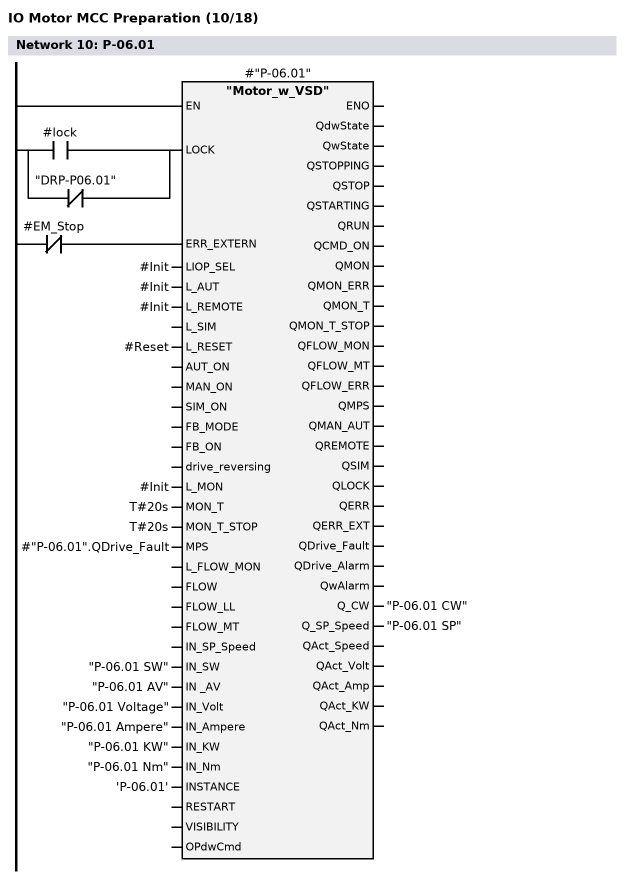
   RUNG wire#powerrail
      #"P-06.01"(LOCK := wire#w1, ERR_EXTERN := wire#w2, LIOP_SEL := #Init, L_AUT := #Init, L_REMOTE := #Init, L_SIM :=, L_RESET := #Reset, AUT_ON :=, MAN_ON :=, SIM_ON :=, FB_MODE :=, FB_ON :=, drive_reversing :=, L_MON := #Init, MON_T := T#20s, MON_T_STOP := T#20s, MPS := #"P-06.01".QDrive_Fault, L_FLOW_MON :=, FLOW :=, FLOW_LL :=, FLOW_MT :=, IN_SP_Speed :=, IN_SW := "P-06.01 SW", "IN _AV" := "P-06.01 AV", IN_Volt := "P-06.01 Voltage", IN_Ampere := "P-06.01 Ampere", IN_KW := "P-06.01 KW", IN_Nm := "P-06.01 Nm", INSTANCE := 'P-06.01', RESTART :=, VISIBILITY :=, OPdwCmd :=, QdwState =>, QwState =>, QSTOPPING =>, QSTOP =>, QSTARTING =>, QRUN =>, QCMD_ON =>, QMON =>, QMON_ERR =>, QMON_T =>, QMON_T_STOP =>, QFLOW_MON =>, QFLOW_MT =>, QFLOW_ERR =>, QMPS =>, QMAN_AUT =>, QREMOTE =>, QSIM =>, QLOCK =>, QERR =>, QERR_EXT =>, QDrive_Fault =>, QDrive_Alarm =>, QwAlarm =>, Q_CW => "P-06.01 CW", Q_SP_Speed => "P-06.01 SP", QAct_Speed =>, QAct_Volt =>, QAct_Amp =>, QAct_KW =>, QAct_Nm =>)
   END_RUNG
   RUNG wire#powerrail
      Contact( #lock )
   END_RUNG wire#w1
   RUNG wire#powerrail
      I_Contact( "DRP-P06.01" )
   END_RUNG wire#w1
   RUNG wire#powerrail
      I_Contact( #EM_Stop )
   END_RUNG wire#w2
   // the same network as SCL:
   #"P-06.01"(LOCK := #lock OR NOT "DRP-P06.01",   // "Motor_w_VSD"
              ERR_EXTERN := NOT #EM_Stop,
              LIOP_SEL := #Init,
              L_AUT := #Init,
              L_REMOTE := #Init,
              L_RESET := #Reset,
              L_MON := #Init,
              MON_T := T#20s,
              MON_T_STOP := T#20s,
              MPS := #"P-06.01".QDrive_Fault,
              IN_SW := "P-06.01 SW",
              "IN _AV" := "P-06.01 AV",
              IN_Volt := "P-06.01 Voltage",
              IN_Ampere := "P-06.01 Ampere",
              IN_KW := "P-06.01 KW",
              IN_Nm := "P-06.01 Nm",
              INSTANCE := 'P-06.01',
              Q_CW => "P-06.01 CW",
              Q_SP_Speed => "P-06.01 SP");
END_REGION

REGION Network 11: P-07.01
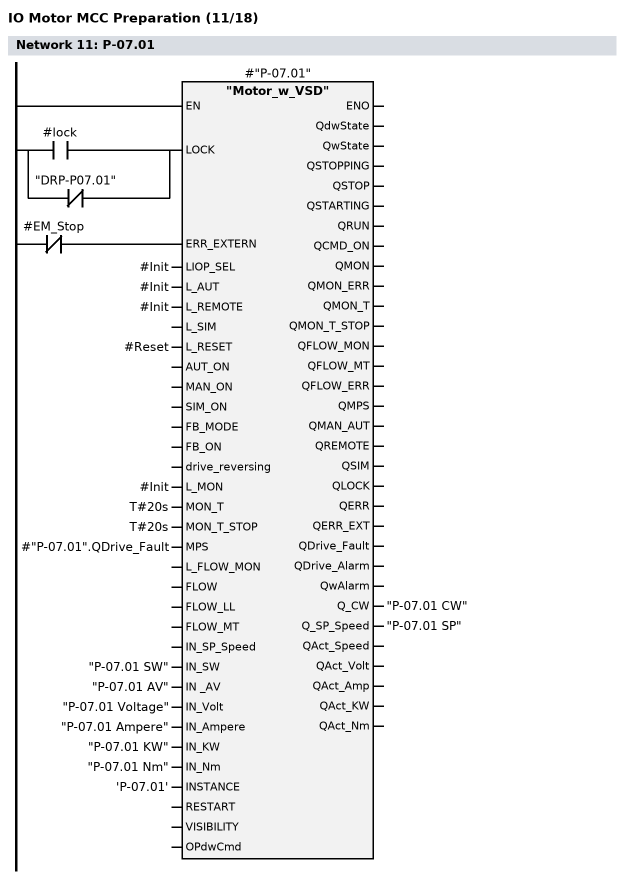
   RUNG wire#powerrail
      #"P-07.01"(LOCK := wire#w1, ERR_EXTERN := wire#w2, LIOP_SEL := #Init, L_AUT := #Init, L_REMOTE := #Init, L_SIM :=, L_RESET := #Reset, AUT_ON :=, MAN_ON :=, SIM_ON :=, FB_MODE :=, FB_ON :=, drive_reversing :=, L_MON := #Init, MON_T := T#20s, MON_T_STOP := T#20s, MPS := #"P-07.01".QDrive_Fault, L_FLOW_MON :=, FLOW :=, FLOW_LL :=, FLOW_MT :=, IN_SP_Speed :=, IN_SW := "P-07.01 SW", "IN _AV" := "P-07.01 AV", IN_Volt := "P-07.01 Voltage", IN_Ampere := "P-07.01 Ampere", IN_KW := "P-07.01 KW", IN_Nm := "P-07.01 Nm", INSTANCE := 'P-07.01', RESTART :=, VISIBILITY :=, OPdwCmd :=, QdwState =>, QwState =>, QSTOPPING =>, QSTOP =>, QSTARTING =>, QRUN =>, QCMD_ON =>, QMON =>, QMON_ERR =>, QMON_T =>, QMON_T_STOP =>, QFLOW_MON =>, QFLOW_MT =>, QFLOW_ERR =>, QMPS =>, QMAN_AUT =>, QREMOTE =>, QSIM =>, QLOCK =>, QERR =>, QERR_EXT =>, QDrive_Fault =>, QDrive_Alarm =>, QwAlarm =>, Q_CW => "P-07.01 CW", Q_SP_Speed => "P-07.01 SP", QAct_Speed =>, QAct_Volt =>, QAct_Amp =>, QAct_KW =>, QAct_Nm =>)
   END_RUNG
   RUNG wire#powerrail
      Contact( #lock )
   END_RUNG wire#w1
   RUNG wire#powerrail
      I_Contact( "DRP-P07.01" )
   END_RUNG wire#w1
   RUNG wire#powerrail
      I_Contact( #EM_Stop )
   END_RUNG wire#w2
   // the same network as SCL:
   #"P-07.01"(LOCK := #lock OR NOT "DRP-P07.01",   // "Motor_w_VSD"
              ERR_EXTERN := NOT #EM_Stop,
              LIOP_SEL := #Init,
              L_AUT := #Init,
              L_REMOTE := #Init,
              L_RESET := #Reset,
              L_MON := #Init,
              MON_T := T#20s,
              MON_T_STOP := T#20s,
              MPS := #"P-07.01".QDrive_Fault,
              IN_SW := "P-07.01 SW",
              "IN _AV" := "P-07.01 AV",
              IN_Volt := "P-07.01 Voltage",
              IN_Ampere := "P-07.01 Ampere",
              IN_KW := "P-07.01 KW",
              IN_Nm := "P-07.01 Nm",
              INSTANCE := 'P-07.01',
              Q_CW => "P-07.01 CW",
              Q_SP_Speed => "P-07.01 SP");
END_REGION

REGION Network 12: P-08.01
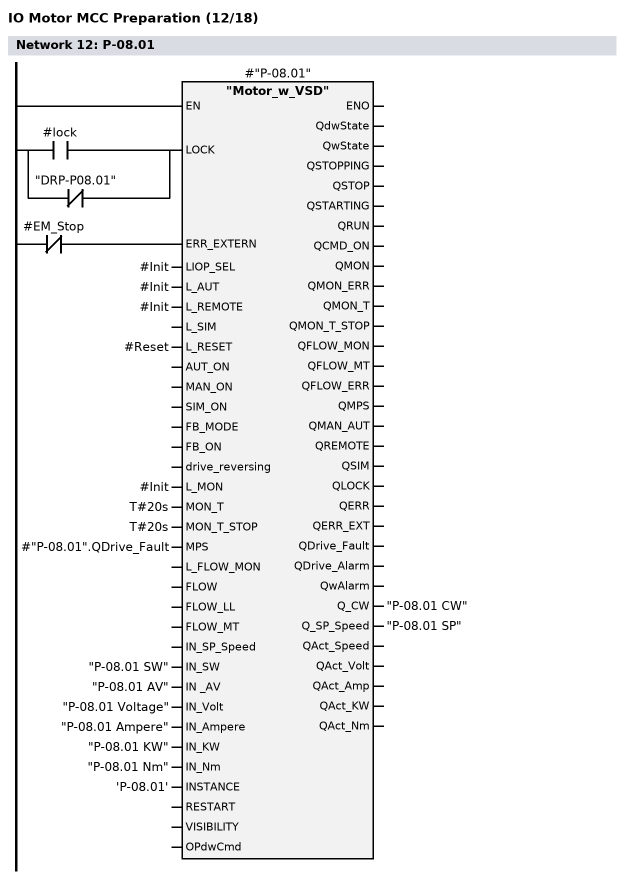
   RUNG wire#powerrail
      #"P-08.01"(LOCK := wire#w1, ERR_EXTERN := wire#w2, LIOP_SEL := #Init, L_AUT := #Init, L_REMOTE := #Init, L_SIM :=, L_RESET := #Reset, AUT_ON :=, MAN_ON :=, SIM_ON :=, FB_MODE :=, FB_ON :=, drive_reversing :=, L_MON := #Init, MON_T := T#20s, MON_T_STOP := T#20s, MPS := #"P-08.01".QDrive_Fault, L_FLOW_MON :=, FLOW :=, FLOW_LL :=, FLOW_MT :=, IN_SP_Speed :=, IN_SW := "P-08.01 SW", "IN _AV" := "P-08.01 AV", IN_Volt := "P-08.01 Voltage", IN_Ampere := "P-08.01 Ampere", IN_KW := "P-08.01 KW", IN_Nm := "P-08.01 Nm", INSTANCE := 'P-08.01', RESTART :=, VISIBILITY :=, OPdwCmd :=, QdwState =>, QwState =>, QSTOPPING =>, QSTOP =>, QSTARTING =>, QRUN =>, QCMD_ON =>, QMON =>, QMON_ERR =>, QMON_T =>, QMON_T_STOP =>, QFLOW_MON =>, QFLOW_MT =>, QFLOW_ERR =>, QMPS =>, QMAN_AUT =>, QREMOTE =>, QSIM =>, QLOCK =>, QERR =>, QERR_EXT =>, QDrive_Fault =>, QDrive_Alarm =>, QwAlarm =>, Q_CW => "P-08.01 CW", Q_SP_Speed => "P-08.01 SP", QAct_Speed =>, QAct_Volt =>, QAct_Amp =>, QAct_KW =>, QAct_Nm =>)
   END_RUNG
   RUNG wire#powerrail
      Contact( #lock )
   END_RUNG wire#w1
   RUNG wire#powerrail
      I_Contact( "DRP-P08.01" )
   END_RUNG wire#w1
   RUNG wire#powerrail
      I_Contact( #EM_Stop )
   END_RUNG wire#w2
   // the same network as SCL:
   #"P-08.01"(LOCK := #lock OR NOT "DRP-P08.01",   // "Motor_w_VSD"
              ERR_EXTERN := NOT #EM_Stop,
              LIOP_SEL := #Init,
              L_AUT := #Init,
              L_REMOTE := #Init,
              L_RESET := #Reset,
              L_MON := #Init,
              MON_T := T#20s,
              MON_T_STOP := T#20s,
              MPS := #"P-08.01".QDrive_Fault,
              IN_SW := "P-08.01 SW",
              "IN _AV" := "P-08.01 AV",
              IN_Volt := "P-08.01 Voltage",
              IN_Ampere := "P-08.01 Ampere",
              IN_KW := "P-08.01 KW",
              IN_Nm := "P-08.01 Nm",
              INSTANCE := 'P-08.01',
              Q_CW => "P-08.01 CW",
              Q_SP_Speed => "P-08.01 SP");
END_REGION

REGION Network 13: P-08.02
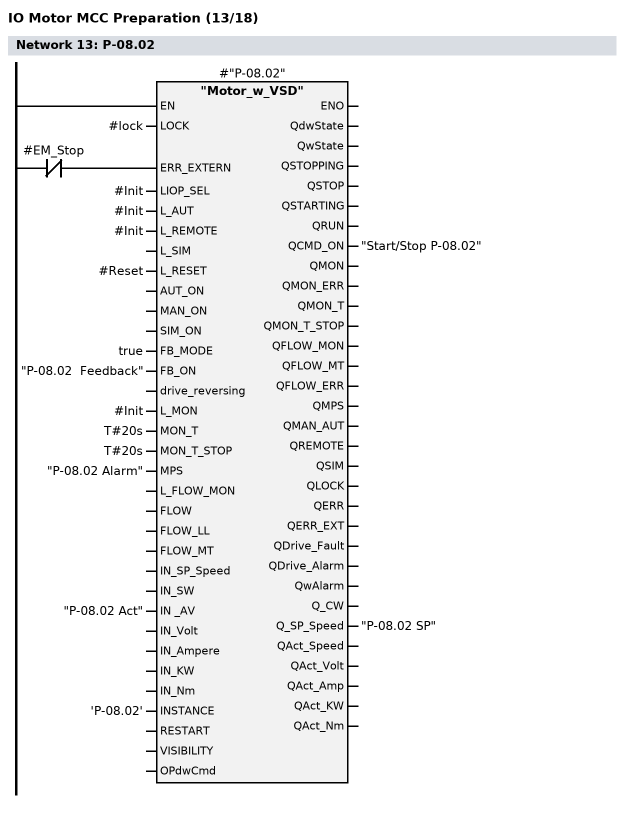
   RUNG wire#powerrail
      #"P-08.02"(ERR_EXTERN := wire#w1, LOCK := #lock, LIOP_SEL := #Init, L_AUT := #Init, L_REMOTE := #Init, L_SIM :=, L_RESET := #Reset, AUT_ON :=, MAN_ON :=, SIM_ON :=, FB_MODE := true, FB_ON := "P-08.02  Feedback", drive_reversing :=, L_MON := #Init, MON_T := T#20s, MON_T_STOP := T#20s, MPS := "P-08.02 Alarm", L_FLOW_MON :=, FLOW :=, FLOW_LL :=, FLOW_MT :=, IN_SP_Speed :=, IN_SW :=, "IN _AV" := "P-08.02 Act", IN_Volt :=, IN_Ampere :=, IN_KW :=, IN_Nm :=, INSTANCE := 'P-08.02', RESTART :=, VISIBILITY :=, OPdwCmd :=, QdwState =>, QwState =>, QSTOPPING =>, QSTOP =>, QSTARTING =>, QRUN =>, QCMD_ON => "Start/Stop P-08.02", QMON =>, QMON_ERR =>, QMON_T =>, QMON_T_STOP =>, QFLOW_MON =>, QFLOW_MT =>, QFLOW_ERR =>, QMPS =>, QMAN_AUT =>, QREMOTE =>, QSIM =>, QLOCK =>, QERR =>, QERR_EXT =>, QDrive_Fault =>, QDrive_Alarm =>, QwAlarm =>, Q_CW =>, Q_SP_Speed => "P-08.02 SP", QAct_Speed =>, QAct_Volt =>, QAct_Amp =>, QAct_KW =>, QAct_Nm =>)
   END_RUNG
   RUNG wire#powerrail
      I_Contact( #EM_Stop )
   END_RUNG wire#w1
   // the same network as SCL:
   #"P-08.02"(LOCK := #lock,   // "Motor_w_VSD"
              ERR_EXTERN := NOT #EM_Stop,
              LIOP_SEL := #Init,
              L_AUT := #Init,
              L_REMOTE := #Init,
              L_RESET := #Reset,
              FB_MODE := true,
              FB_ON := "P-08.02  Feedback",
              L_MON := #Init,
              MON_T := T#20s,
              MON_T_STOP := T#20s,
              MPS := "P-08.02 Alarm",
              "IN _AV" := "P-08.02 Act",
              INSTANCE := 'P-08.02',
              QCMD_ON => "Start/Stop P-08.02",
              Q_SP_Speed => "P-08.02 SP");
END_REGION

REGION Network 14: XA-09.01
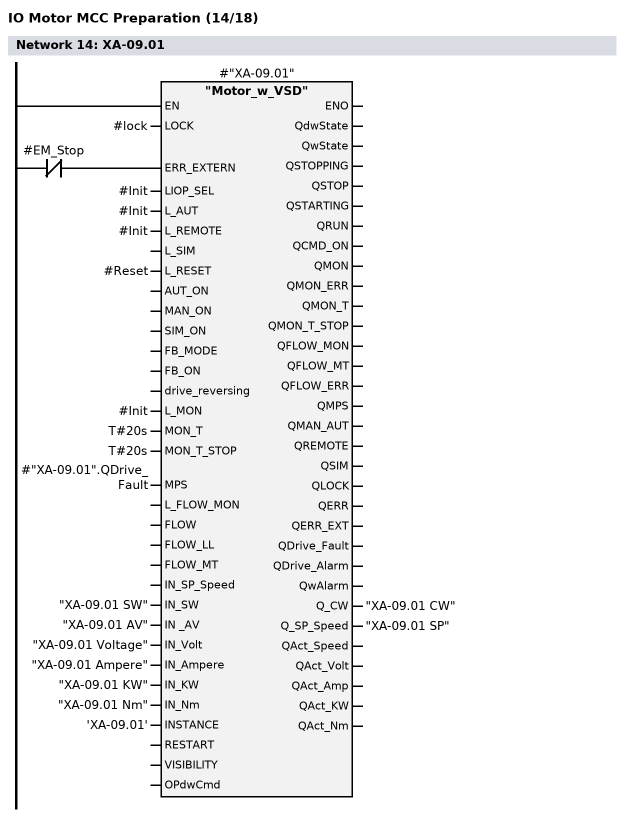
   RUNG wire#powerrail
      #"XA-09.01"(ERR_EXTERN := wire#w1, LOCK := #lock, LIOP_SEL := #Init, L_AUT := #Init, L_REMOTE := #Init, L_SIM :=, L_RESET := #Reset, AUT_ON :=, MAN_ON :=, SIM_ON :=, FB_MODE :=, FB_ON :=, drive_reversing :=, L_MON := #Init, MON_T := T#20s, MON_T_STOP := T#20s, MPS := #"XA-09.01".QDrive_Fault, L_FLOW_MON :=, FLOW :=, FLOW_LL :=, FLOW_MT :=, IN_SP_Speed :=, IN_SW := "XA-09.01 SW", "IN _AV" := "XA-09.01 AV", IN_Volt := "XA-09.01 Voltage", IN_Ampere := "XA-09.01 Ampere", IN_KW := "XA-09.01 KW", IN_Nm := "XA-09.01 Nm", INSTANCE := 'XA-09.01', RESTART :=, VISIBILITY :=, OPdwCmd :=, QdwState =>, QwState =>, QSTOPPING =>, QSTOP =>, QSTARTING =>, QRUN =>, QCMD_ON =>, QMON =>, QMON_ERR =>, QMON_T =>, QMON_T_STOP =>, QFLOW_MON =>, QFLOW_MT =>, QFLOW_ERR =>, QMPS =>, QMAN_AUT =>, QREMOTE =>, QSIM =>, QLOCK =>, QERR =>, QERR_EXT =>, QDrive_Fault =>, QDrive_Alarm =>, QwAlarm =>, Q_CW => "XA-09.01 CW", Q_SP_Speed => "XA-09.01 SP", QAct_Speed =>, QAct_Volt =>, QAct_Amp =>, QAct_KW =>, QAct_Nm =>)
   END_RUNG
   RUNG wire#powerrail
      I_Contact( #EM_Stop )
   END_RUNG wire#w1
   // the same network as SCL:
   #"XA-09.01"(LOCK := #lock,   // "Motor_w_VSD"
               ERR_EXTERN := NOT #EM_Stop,
               LIOP_SEL := #Init,
               L_AUT := #Init,
               L_REMOTE := #Init,
               L_RESET := #Reset,
               L_MON := #Init,
               MON_T := T#20s,
               MON_T_STOP := T#20s,
               MPS := #"XA-09.01".QDrive_Fault,
               IN_SW := "XA-09.01 SW",
               "IN _AV" := "XA-09.01 AV",
               IN_Volt := "XA-09.01 Voltage",
               IN_Ampere := "XA-09.01 Ampere",
               IN_KW := "XA-09.01 KW",
               IN_Nm := "XA-09.01 Nm",
               INSTANCE := 'XA-09.01',
               Q_CW => "XA-09.01 CW",
               Q_SP_Speed => "XA-09.01 SP");
END_REGION

REGION Network 15: P-09.01
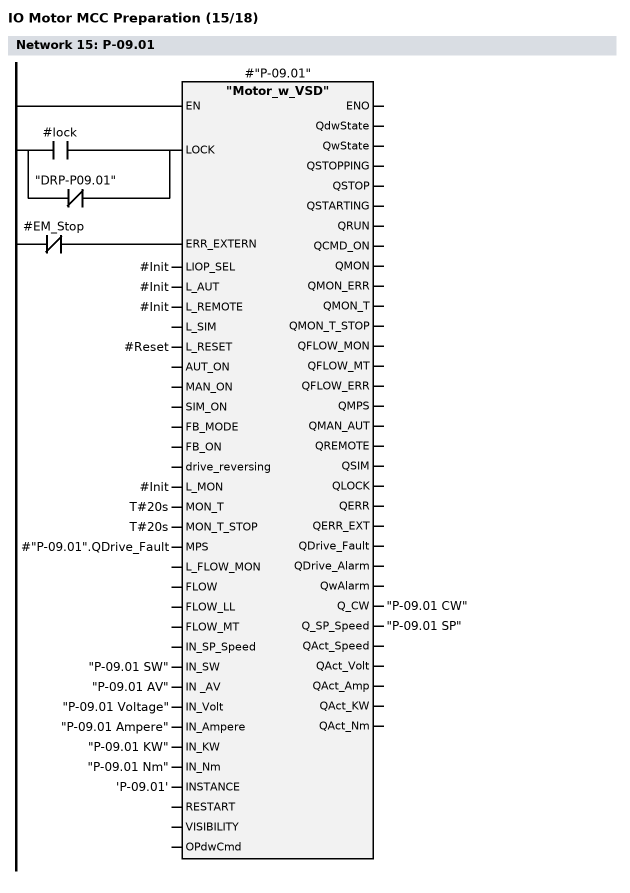
   RUNG wire#powerrail
      #"P-09.01"(LOCK := wire#w1, ERR_EXTERN := wire#w2, LIOP_SEL := #Init, L_AUT := #Init, L_REMOTE := #Init, L_SIM :=, L_RESET := #Reset, AUT_ON :=, MAN_ON :=, SIM_ON :=, FB_MODE :=, FB_ON :=, drive_reversing :=, L_MON := #Init, MON_T := T#20s, MON_T_STOP := T#20s, MPS := #"P-09.01".QDrive_Fault, L_FLOW_MON :=, FLOW :=, FLOW_LL :=, FLOW_MT :=, IN_SP_Speed :=, IN_SW := "P-09.01 SW", "IN _AV" := "P-09.01 AV", IN_Volt := "P-09.01 Voltage", IN_Ampere := "P-09.01 Ampere", IN_KW := "P-09.01 KW", IN_Nm := "P-09.01 Nm", INSTANCE := 'P-09.01', RESTART :=, VISIBILITY :=, OPdwCmd :=, QdwState =>, QwState =>, QSTOPPING =>, QSTOP =>, QSTARTING =>, QRUN =>, QCMD_ON =>, QMON =>, QMON_ERR =>, QMON_T =>, QMON_T_STOP =>, QFLOW_MON =>, QFLOW_MT =>, QFLOW_ERR =>, QMPS =>, QMAN_AUT =>, QREMOTE =>, QSIM =>, QLOCK =>, QERR =>, QERR_EXT =>, QDrive_Fault =>, QDrive_Alarm =>, QwAlarm =>, Q_CW => "P-09.01 CW", Q_SP_Speed => "P-09.01 SP", QAct_Speed =>, QAct_Volt =>, QAct_Amp =>, QAct_KW =>, QAct_Nm =>)
   END_RUNG
   RUNG wire#powerrail
      Contact( #lock )
   END_RUNG wire#w1
   RUNG wire#powerrail
      I_Contact( "DRP-P09.01" )
   END_RUNG wire#w1
   RUNG wire#powerrail
      I_Contact( #EM_Stop )
   END_RUNG wire#w2
   // the same network as SCL:
   #"P-09.01"(LOCK := #lock OR NOT "DRP-P09.01",   // "Motor_w_VSD"
              ERR_EXTERN := NOT #EM_Stop,
              LIOP_SEL := #Init,
              L_AUT := #Init,
              L_REMOTE := #Init,
              L_RESET := #Reset,
              L_MON := #Init,
              MON_T := T#20s,
              MON_T_STOP := T#20s,
              MPS := #"P-09.01".QDrive_Fault,
              IN_SW := "P-09.01 SW",
              "IN _AV" := "P-09.01 AV",
              IN_Volt := "P-09.01 Voltage",
              IN_Ampere := "P-09.01 Ampere",
              IN_KW := "P-09.01 KW",
              IN_Nm := "P-09.01 Nm",
              INSTANCE := 'P-09.01',
              Q_CW => "P-09.01 CW",
              Q_SP_Speed => "P-09.01 SP");
END_REGION

REGION Network 16: P-09.03 DOL
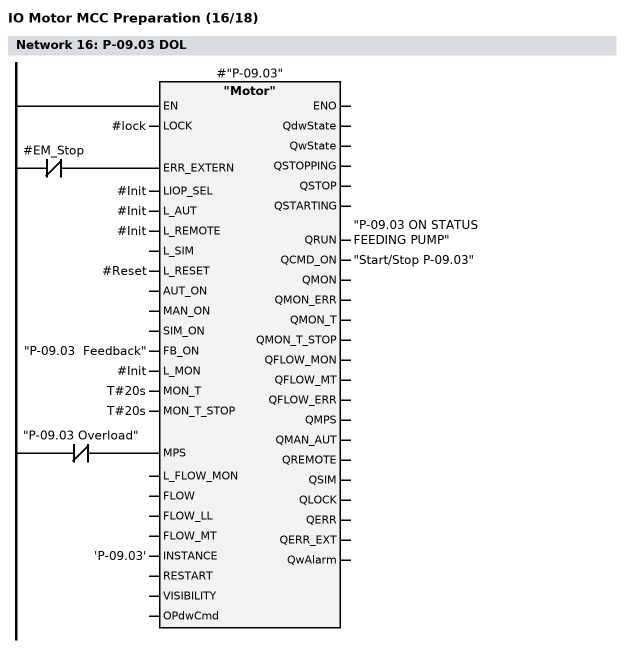
   RUNG wire#powerrail
      #"P-09.03"(ERR_EXTERN := wire#w1, MPS := wire#w2, LOCK := #lock, LIOP_SEL := #Init, L_AUT := #Init, L_REMOTE := #Init, L_SIM :=, L_RESET := #Reset, AUT_ON :=, MAN_ON :=, SIM_ON :=, FB_ON := "P-09.03  Feedback", L_MON := #Init, MON_T := T#20s, MON_T_STOP := T#20s, L_FLOW_MON :=, FLOW :=, FLOW_LL :=, FLOW_MT :=, INSTANCE := 'P-09.03', RESTART :=, VISIBILITY :=, OPdwCmd :=, QdwState =>, QwState =>, QSTOPPING =>, QSTOP =>, QSTARTING =>, QRUN => "P-09.03 ON STATUS FEEDING PUMP", QCMD_ON => "Start/Stop P-09.03", QMON =>, QMON_ERR =>, QMON_T =>, QMON_T_STOP =>, QFLOW_MON =>, QFLOW_MT =>, QFLOW_ERR =>, QMPS =>, QMAN_AUT =>, QREMOTE =>, QSIM =>, QLOCK =>, QERR =>, QERR_EXT =>, QwAlarm =>)
   END_RUNG
   RUNG wire#powerrail
      I_Contact( #EM_Stop )
   END_RUNG wire#w1
   RUNG wire#powerrail
      I_Contact( "P-09.03 Overload" )
   END_RUNG wire#w2
   // the same network as SCL:
   #"P-09.03"(LOCK := #lock,   // "Motor"
              ERR_EXTERN := NOT #EM_Stop,
              LIOP_SEL := #Init,
              L_AUT := #Init,
              L_REMOTE := #Init,
              L_RESET := #Reset,
              FB_ON := "P-09.03  Feedback",
              L_MON := #Init,
              MON_T := T#20s,
              MON_T_STOP := T#20s,
              MPS := NOT "P-09.03 Overload",
              INSTANCE := 'P-09.03',
              QRUN => "P-09.03 ON STATUS FEEDING PUMP",
              QCMD_ON => "Start/Stop P-09.03");
END_REGION

REGION Network 17: P-10.01
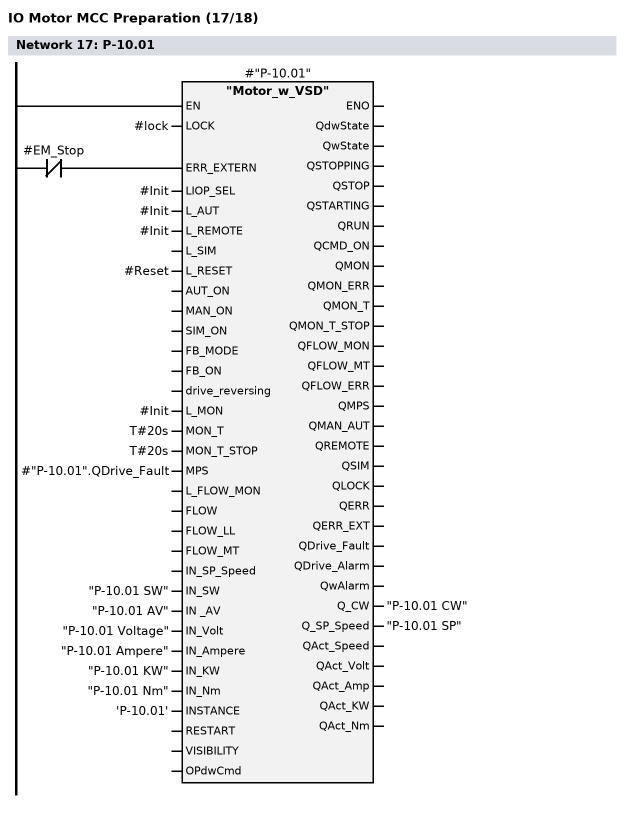
   RUNG wire#powerrail
      #"P-10.01"(ERR_EXTERN := wire#w1, LOCK := #lock, LIOP_SEL := #Init, L_AUT := #Init, L_REMOTE := #Init, L_SIM :=, L_RESET := #Reset, AUT_ON :=, MAN_ON :=, SIM_ON :=, FB_MODE :=, FB_ON :=, drive_reversing :=, L_MON := #Init, MON_T := T#20s, MON_T_STOP := T#20s, MPS := #"P-10.01".QDrive_Fault, L_FLOW_MON :=, FLOW :=, FLOW_LL :=, FLOW_MT :=, IN_SP_Speed :=, IN_SW := "P-10.01 SW", "IN _AV" := "P-10.01 AV", IN_Volt := "P-10.01 Voltage", IN_Ampere := "P-10.01 Ampere", IN_KW := "P-10.01 KW", IN_Nm := "P-10.01 Nm", INSTANCE := 'P-10.01', RESTART :=, VISIBILITY :=, OPdwCmd :=, QdwState =>, QwState =>, QSTOPPING =>, QSTOP =>, QSTARTING =>, QRUN =>, QCMD_ON =>, QMON =>, QMON_ERR =>, QMON_T =>, QMON_T_STOP =>, QFLOW_MON =>, QFLOW_MT =>, QFLOW_ERR =>, QMPS =>, QMAN_AUT =>, QREMOTE =>, QSIM =>, QLOCK =>, QERR =>, QERR_EXT =>, QDrive_Fault =>, QDrive_Alarm =>, QwAlarm =>, Q_CW => "P-10.01 CW", Q_SP_Speed => "P-10.01 SP", QAct_Speed =>, QAct_Volt =>, QAct_Amp =>, QAct_KW =>, QAct_Nm =>)
   END_RUNG
   RUNG wire#powerrail
      I_Contact( #EM_Stop )
   END_RUNG wire#w1
   // the same network as SCL:
   #"P-10.01"(LOCK := #lock,   // "Motor_w_VSD"
              ERR_EXTERN := NOT #EM_Stop,
              LIOP_SEL := #Init,
              L_AUT := #Init,
              L_REMOTE := #Init,
              L_RESET := #Reset,
              L_MON := #Init,
              MON_T := T#20s,
              MON_T_STOP := T#20s,
              MPS := #"P-10.01".QDrive_Fault,
              IN_SW := "P-10.01 SW",
              "IN _AV" := "P-10.01 AV",
              IN_Volt := "P-10.01 Voltage",
              IN_Ampere := "P-10.01 Ampere",
              IN_KW := "P-10.01 KW",
              IN_Nm := "P-10.01 Nm",
              INSTANCE := 'P-10.01',
              Q_CW => "P-10.01 CW",
              Q_SP_Speed => "P-10.01 SP");
END_REGION

REGION Network 18: P-51.01
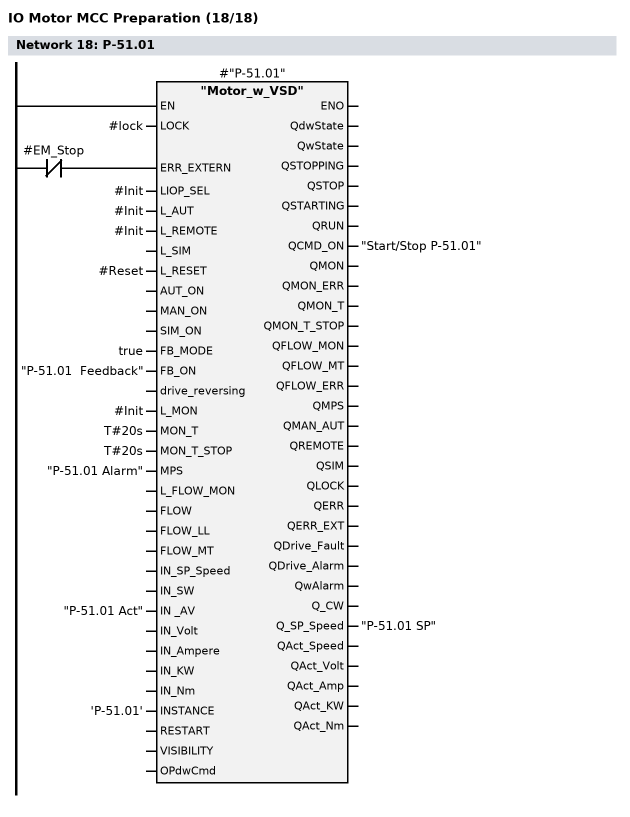
   RUNG wire#powerrail
      #"P-51.01"(ERR_EXTERN := wire#w1, LOCK := #lock, LIOP_SEL := #Init, L_AUT := #Init, L_REMOTE := #Init, L_SIM :=, L_RESET := #Reset, AUT_ON :=, MAN_ON :=, SIM_ON :=, FB_MODE := true, FB_ON := "P-51.01  Feedback", drive_reversing :=, L_MON := #Init, MON_T := T#20s, MON_T_STOP := T#20s, MPS := "P-51.01 Alarm", L_FLOW_MON :=, FLOW :=, FLOW_LL :=, FLOW_MT :=, IN_SP_Speed :=, IN_SW :=, "IN _AV" := "P-51.01 Act", IN_Volt :=, IN_Ampere :=, IN_KW :=, IN_Nm :=, INSTANCE := 'P-51.01', RESTART :=, VISIBILITY :=, OPdwCmd :=, QdwState =>, QwState =>, QSTOPPING =>, QSTOP =>, QSTARTING =>, QRUN =>, QCMD_ON => "Start/Stop P-51.01", QMON =>, QMON_ERR =>, QMON_T =>, QMON_T_STOP =>, QFLOW_MON =>, QFLOW_MT =>, QFLOW_ERR =>, QMPS =>, QMAN_AUT =>, QREMOTE =>, QSIM =>, QLOCK =>, QERR =>, QERR_EXT =>, QDrive_Fault =>, QDrive_Alarm =>, QwAlarm =>, Q_CW =>, Q_SP_Speed => "P-51.01 SP", QAct_Speed =>, QAct_Volt =>, QAct_Amp =>, QAct_KW =>, QAct_Nm =>)
   END_RUNG
   RUNG wire#powerrail
      I_Contact( #EM_Stop )
   END_RUNG wire#w1
   // the same network as SCL:
   #"P-51.01"(LOCK := #lock,   // "Motor_w_VSD"
              ERR_EXTERN := NOT #EM_Stop,
              LIOP_SEL := #Init,
              L_AUT := #Init,
              L_REMOTE := #Init,
              L_RESET := #Reset,
              FB_MODE := true,
              FB_ON := "P-51.01  Feedback",
              L_MON := #Init,
              MON_T := T#20s,
              MON_T_STOP := T#20s,
              MPS := "P-51.01 Alarm",
              "IN _AV" := "P-51.01 Act",
              INSTANCE := 'P-51.01',
              QCMD_ON => "Start/Stop P-51.01",
              Q_SP_Speed => "P-51.01 SP");
END_REGION
END_FUNCTION_BLOCK

FUNCTION_BLOCK "Motor_w_VSD"
TITLE = Motor
{ S7_Optimized_Access := 'FALSE' }
AUTHOR : IW
VERSION : 0.1
//Interface FB for a motor with Danfoss FC Profil
   VAR_INPUT 
      LOCK : Bool;   // 1 = Interlock active
      ERR_EXTERN : Bool;   // 1 = External error arised
      LIOP_SEL : Bool;   // 0 = Operator; 1 = Linking
      L_AUT : Bool;   // 0 = Manual; 1 = Automatic
      L_REMOTE : Bool;   // 0 = Local; 1 = Remote
      L_SIM : Bool;   // 0 = Normal; 1 = Simulation
      L_RESET : Bool;   // 1 = Reset error peripherie
      AUT_ON : Bool;   // 1 = CMD ON Automatic
      MAN_ON : Bool;   // 1 = CMD ON Manual
      SIM_ON : Bool;   // 1 = CMD ON Simulation
      FB_MODE : Bool;   // 0 = FB Run from communication ,1 = FB_ON
      FB_ON : Bool;   // 1 = Feedback Motor ON
      drive_reversing : Bool;
      L_MON : Bool;   // 1 = Monitoring ON
      MON_T : Time := t#5s;   // Monitoring starting time in process mode
      MON_T_STOP : Time := t#5s;   // Monitoring stopping time in process mode
      MPS : Bool;   // 1 = Motor protection switch ON
      L_FLOW_MON : Bool;   // 1 = Monitoring flow
      FLOW : Real;   // Current flow
      FLOW_LL : Real := 5.0;   // Low level flow
      FLOW_MT : Time := t#8s;   // Delay of monitoring lower flow
      IN_SP_Speed : Real;   // Setpoint Speed in Percen
      IN_SW : Word;   // IN Status word from Drive
      "IN _AV" : Int;   // IN Actual Speed from Drive
      IN_Volt : Int;   // IN Actual Voltage
      IN_Ampere : Int;   // IN Actual Ampere
      IN_KW : Int;   // IN Actual KW
      IN_Nm : Int;   // IN Actual Torque
      INSTANCE : String := 'Motor_001';   // Filter attribute for message view, also used for labelling
      RESTART : Bool;   // 1 = Initialize FB at startup (first cycle of PLC)
   END_VAR

   VAR_OUTPUT 
      QdwState : DWord;   // Status HMI
      QwState : Int;   // Motor: 0 = Stop; 1 = Starting; 2 = Run; 3 = Stopping
      QSTOPPING : Bool;   // 1 = Stopping
      QSTOP : Bool;   // 1 = Stop
      QSTARTING : Bool;   // 1 = Starting
      QRUN : Bool;   // 1 = Run
      QCMD_ON : Bool;   // 0 = Stop; 1 = Start (automatic & manual mode)
      QMON : Bool;   // 1 = Monitoring is ON
      QMON_ERR : Bool;   // 1 = Monitoring errror
      QMON_T : Time;   // Expierd starting time in process mode
      QMON_T_STOP : Time;   // Expierd stopping time in process mode
      QFLOW_MON : Bool;   // 1 = Flow monitoring is ON
      QFLOW_MT : Time;   // Expiered delay of monitoring lower flow
      QFLOW_ERR : Bool;   // 1 = Error flow monitoring
      QMPS : Bool;   // 1 = Motor protecting switch
      QMAN_AUT : Bool;   // 0 = Manual; 1 = Automatic
      QREMOTE : Bool;   // 0 = Local; 1 = Remote
      QSIM : Bool;   // 0 = Normal; 1 = Simulation
      QLOCK : Bool;   // 1 = Interlock is active
      QERR : Bool;   // 1 = Common error
      QERR_EXT : Bool;   // 1 = External error
      QDrive_Fault : Bool;
      QDrive_Alarm : Bool;
      QwAlarm : Word;   // Bit alarm procedure
      Q_CW : Word;   // Out Control Word for VSD
      Q_SP_Speed : Word;   // Out SP Speed for VSD
      QAct_Speed : Real;   // Drive Actual Speed
      QAct_Volt : Real;   // Drive Actual Voltage
      QAct_Amp : Real;   // Drive Actual Ampere
      QAct_KW : Real;   // Drive Actual KW
      QAct_Nm : Real;   // Drive Actual Torque
   END_VAR

   VAR_IN_OUT 
      VISIBILITY : Byte;   // Bit 0: Tab1 of window; Bit 1: Tab2 of window; ... ; Bit 7: Minimize
      OPdwCmd : DWord;   // Contorl word HMI
   END_VAR

   VAR 
      FB_SIM : Bool;
      SP_SpeedHz : Real;   // setengah dari 100%
      Drive_Actual_Speed : Real;   // Drive Actual Speed in Percen
      Drive_CW : Word;
      Drive_SW : Word;
      SIM_T : Time;
      QSIM_T : Time;
      SIM_T_STOP : Time;
      QSIM_T_STOP : Time;
      QCMD_SIM : Bool;
      OP_RESET : Bool;   // Reset errors
      QFLOW_MON_ACK : Bool;
      OP_VISIBILITY : Byte;   // Bit 0: Tab1 of window; Bit 1: Tab2 of window; ... ; Bit 7: Minimize
      VISIBILITY_OLD : Byte;   // Save last status of VISIBILITY
      QFB_RUN : Bool;
      Drive_FB_ON : Bool;   // Drive_Running
      Drive_Fault : Bool;   // Drive_Fault Active
      Drive_Alarm : Bool;   // Drive_Alarm Active
      Drive_OK : Bool;
      SE_L_RESET_LINK : Bool;   // Signal edge for the reset input from linking
      SE_L_RESET_LINK_COND : Bool;   // Condition of signal edge
      SE_L_RESET_OP : Bool;   // Signal edge for the reset input from operator
      TSTARTING {InstructionName := 'TON_TIME'; LibVersion := '1.0'} : TON_TIME;
      TSTOPPING {InstructionName := 'TON_TIME'; LibVersion := '1.0'} : TON_TIME;
      TFLOW {InstructionName := 'TON_TIME'; LibVersion := '1.0'} : TON_TIME;
      TSTARTING_SIM {InstructionName := 'TON_TIME'; LibVersion := '1.0'} : TON_TIME;
      TSTOPPING_SIM {InstructionName := 'TON_TIME'; LibVersion := '1.0'} : TON_TIME;
   END_VAR

   VAR_TEMP 
      CON_ERR : Bool;   // Error in motor condition
      MON_ERR_STARTING : Bool;   // Monitoring error for starting motor in process mode
      MON_ERR_STOPPING : Bool;   // Monitoring error for stopping motor in process mode
      MON_SIM_STARTING : Bool;   // Monitoring error for starting motor in simulation mode
      MON_SIM_STOPPING : Bool;   // Monitoring error for stopping motor in simulation mode
      FB_ERR : Bool;   // Feedback error in process mode
      MON_ERR_FLOW2 : Bool;
      START_FLOW_TIME2 : Bool;
      START_FLOW_TIME : Bool;   // Start Signal of delay time for flow
      MON_ERR_FLOW : Bool;   // Monitoring error for flow
   END_VAR


BEGIN
	(********************************
	           Start up
	*********************************)
	IF #RESTART= true THEN
	  // Restart case
	  #QCMD_ON:= false;
	  #QSTOP:=true;
	  #QSTOPPING:=false;
	  #QRUN:=false;
	  #QSTARTING:=false;
	  #VISIBILITY:=0;
	  #OPdwCmd:=0;
	ELSE
	  // Normal case
	  
	  (******************************************
	    Network 1: Operating mode: manual/automatic
	    Vaiable: OPdwCmd  Bit:  16  =  Manual
	    Vaiable: OPdwCmd  Bit:  17  =  Automatic
	  *******************************************)
	  IF (#LIOP_SEL=true AND #L_AUT=true) OR (#OPdwCmd.%X17=true AND #LIOP_SEL=false) THEN
	    #QMAN_AUT:=true;
	    #OPdwCmd.%X16:=false;
	    #OPdwCmd.%X17:=false;
	  ELSIF (#LIOP_SEL=true AND #L_AUT=false) OR (#OPdwCmd.%X16=true AND #LIOP_SEL=false) THEN
	    #QMAN_AUT:= false;
	    #OPdwCmd.%X16:=false;
	    #OPdwCmd.%X17:=false;
	  END_IF;
	  
	  (******************************************
	    Network 2: Control mode: local/remote
	    Vaiable: OPdwCmd  Bit:  18  =  Local
	    Vaiable: OPdwCmd  Bit:  19  =  Remote
	  *******************************************)
	  IF (#LIOP_SEL=true AND #L_REMOTE=true) OR (#OPdwCmd.%X19=true AND #LIOP_SEL=false) THEN
	    #QREMOTE:=true;
	    #OPdwCmd.%X18:=false;
	    #OPdwCmd.%X19:=false;
	  ELSIF (#LIOP_SEL=true AND #L_REMOTE=false) OR (#OPdwCmd.%X18=true AND #LIOP_SEL=false) THEN
	    #QREMOTE:= false;
	    #OPdwCmd.%X18:=false;
	    #OPdwCmd.%X19:=false;
	  END_IF;
	  
	  (******************************************
	    Network 3: Simulation On/Off
	    Vaiable: OPdwCmd  Bit:  20  =  Process
	    Vaiable: OPdwCmd  Bit:  21  =  Simulation
	  *******************************************)
	  IF (#LIOP_SEL=true AND #L_SIM=true) OR (#OPdwCmd.%X21=true AND #LIOP_SEL=false) THEN
	    #QSIM:=true;
	    #OPdwCmd.%X20:=false;
	    #OPdwCmd.%X21:=false;
	  ELSIF (#LIOP_SEL=true AND #L_SIM=false) OR (#OPdwCmd.%X20=true AND #LIOP_SEL=false) THEN
	    #QSIM:= false;
	    #OPdwCmd.%X20:=false;
	    #OPdwCmd.%X21:=false;
	  END_IF;
	  
	  (*************************************
	    Network 4: Reset Operation
	    Vaiable: OPdwCmd  Bit:  24  =  Reset
	  **************************************)
	  // Rising edge by linking
	  IF #L_RESET=true AND #SE_L_RESET_LINK_COND=false THEN
	    #SE_L_RESET_LINK:=true;
	    #SE_L_RESET_LINK_COND:=true;
	  ELSIF #L_RESET=true AND #SE_L_RESET_LINK_COND=true THEN
	    #SE_L_RESET_LINK:=false;
	  ELSE
	    #SE_L_RESET_LINK_COND:=false;
	  END_IF;
	  // Rising edge by operator
	  IF #OPdwCmd.%X24=true THEN
	    #SE_L_RESET_OP:=true;
	    #OPdwCmd.%X24:=false;
	  ELSE
	    #SE_L_RESET_OP:=false;
	  END_IF;
	  // Reset error #OP_RESET:=((#LIOP_SEL AND #SE_L_RESET_LINK) OR (#SE_L_RESET_OP AND NOT #LIOP_SEL)) AND NOT #LOCK;
	  #OP_RESET:=(#L_RESET) OR (#SE_L_RESET_OP AND NOT #LIOP_SEL) AND NOT #LOCK;
	  
	  (**********************************************
	    Network 5: Monitoring feedback ON/OFF
	    Vaiable: OPdwCmd  Bit:  8  =  Monitoring ON
	    Vaiable: OPdwCmd  Bit:  9  =  Monitoring OFF
	  ***********************************************)
	  IF (#LIOP_SEL=true AND #L_MON=false) OR (#OPdwCmd.%X9=true AND #LIOP_SEL=false)THEN
	    #QMON:=false;
	    #OPdwCmd.%X8:=false;
	    #OPdwCmd.%X9:=false;
	  ELSIF (#LIOP_SEL=true AND #L_MON=true) OR (#OPdwCmd.%X8=true AND #LIOP_SEL=false)THEN
	    #QMON:=true;
	    #OPdwCmd.%X8:=false;
	    #OPdwCmd.%X9:=false;
	  END_IF;
	  
	  (***************************************************
	    Network 6: Monitoring flow ON/OFF
	    Vaiable: OPdwCmd  Bit:  10  =  Monitoring flow ON
	    Vaiable: OPdwCmd  Bit:  11  =  Monitoring flow OFF
	  ****************************************************)
	  IF (#LIOP_SEL=true AND #L_FLOW_MON=false) OR (#OPdwCmd.%X11=true AND #LIOP_SEL=false)THEN
	    #QFLOW_MON:=false;
	    #OPdwCmd.%X10:=false;
	    #OPdwCmd.%X11:=false;
	  ELSIF (#LIOP_SEL=true AND #L_FLOW_MON=true) OR (#OPdwCmd.%X10=true AND #LIOP_SEL=false)THEN
	    #QFLOW_MON:=true;
	    #OPdwCmd.%X10:=false;
	    #OPdwCmd.%X11:=false;
	  END_IF;
	  
	   (**********************************************
	    Network 6: START/STOP Motor
	    Vaiable: OPdwCmd  Bit:  0  =  STOP Motor
	    Vaiable: OPdwCmd  Bit:  1  =  START Motor
	  ***********************************************)
	  IF #QERR=false THEN
	    // No errors occurs
	    IF #QSIM=false THEN
	     // Simulation mode is not active
	      // Automatic/Manual mode
	      IF #QMAN_AUT=true THEN
	        // Automatic mode is active
	        // OPEN/CLOSE valve by linking (AUT_ON)
	        #QCMD_ON:=#AUT_ON;
	        #OPdwCmd.%X0:=false;
	        #OPdwCmd.%X1:=false;
	      ELSE
	       // Automatic mode is not active
	        // Local/Remote mode
	        IF #QREMOTE=false THEN
	          // Local mode is active
	          // OPEN/CLOSE valve by linking (MAN_ON)
	          #QCMD_ON:=#MAN_ON AND NOT #QMAN_AUT;
	          #OPdwCmd.%X0:=false;
	          #OPdwCmd.%X1:=false;
	        ELSE
	         // Remote mode is active
	          // Open valve by operator
	          IF #OPdwCmd.%X1=true THEN
	            #QCMD_ON:=true;
	            #OPdwCmd.%X0:=false;
	            #OPdwCmd.%X1:=false;
	          END_IF;
	          // Close valve by operator
	          IF #OPdwCmd.%X0=true THEN
	            #QCMD_ON:=false;
	            #OPdwCmd.%X0:=false;
	            #OPdwCmd.%X1:=false;
	          END_IF;
	        END_IF;
	      END_IF;
	    ELSE
	      // Local/Remote mode
	      IF #QREMOTE=false THEN
	        // Local mode is active
	          // OPEN/CLOSE valve by linking (SIM_ON)
	          #QCMD_SIM:=#SIM_ON;
	          #OPdwCmd.%X0:=false;
	          #OPdwCmd.%X1:=false;
	      ELSE
	        // Remote mode is active
	          // Open valve by operator
	          IF #OPdwCmd.%X1=true THEN
	            #QCMD_SIM:=true;
	            #OPdwCmd.%X0:=false;
	            #OPdwCmd.%X1:=false;
	          END_IF;
	          // Close valve by operator
	          IF #OPdwCmd.%X0=true THEN
	            #QCMD_SIM:=false;
	            #OPdwCmd.%X0:=false;
	            #OPdwCmd.%X1:=false;
	          END_IF;        
	       END_IF;
	    END_IF;  
	  ELSE
	    // Errors occurs
	    #QCMD_ON:=false;
	    #QCMD_SIM:=false;
	    #OPdwCmd.%X0:=false;
	    #OPdwCmd.%X1:=false;
	  END_IF;
	  
	  (****************************************
	    Network 7: Drive FB_Run
	  *****************************************)
	 // #Drive_FB_ON := #IN_SW.%X2 OR ((#IN_SP_Speed < 5.0)AND #QCMD_ON);
	  #Drive_FB_ON := #IN_SW.%X11 OR ((#IN_SP_Speed < 5.0)AND #QCMD_ON);
	  #QFB_RUN := (#FB_MODE = FALSE AND #Drive_FB_ON) OR (#FB_MODE = TRUE AND (#FB_ON OR ((#IN_SP_Speed < 5.0)AND #QCMD_ON)));
	  (****************************************
	    Network 8: Control signal to the Motor (HMI Status)
	  *****************************************)
	  IF #QERR=false THEN
	    // Motor is stopped
	    IF (((#QFB_RUN=false OR #QMON=false) AND #QSIM=false AND #QCMD_ON=false) OR
	      ((#FB_SIM=false OR #QMON=false) AND #QSIM=true AND #QCMD_SIM=false)) AND #QSTOPPING=true THEN
	      #QSTOP:=true;
	      #QSTOPPING:=false;
	      #QRUN:=false;
	      #QSTARTING := false;
	      #QwState:=0;
	    END_IF;
	    // Motor is stopping
	    IF ((#QSIM=false AND #QCMD_ON=false) OR (#QSIM=true AND #QCMD_SIM=false)) AND (#QRUN=true OR #QSTARTING=true) THEN
	      #QSTOP:=false;
	      #QSTOPPING:=true;
	      #QRUN:=false;
	      #QSTARTING:=false;
	      #QwState:=3;
	    END_IF;
	    // Motor is running 
	    IF (((#QFB_RUN=true OR #QMON=false) AND #QSIM=false AND #QCMD_ON=true) OR
	      ((#FB_SIM=true OR #QMON=false) AND #QSIM=true AND #QCMD_SIM=true)) AND #QSTARTING=true THEN    
	    #QSTOP:=false;
	    #QSTOPPING:=false;
	    #QRUN:=true;
	    #QSTARTING:=false;
	    #QwState:=2;
	    END_IF;
	    // Motor is starting 
	    IF ((#QSIM=false AND #QCMD_ON=true) OR (#QSIM=true AND #QCMD_SIM=true)) AND #QSTOP=true THEN
	    #QSTOP:=false;
	    #QSTOPPING:=false;
	    #QRUN:=false;
	    #QSTARTING:=true;
	    #QwState:=1;
	    END_IF;
	  END_IF;
	  (*******************************************************************
	    Network 9: Drive Control Word
	    *******************************************************************)
	  //Drive_OK
	  #Drive_OK := (#IN_SW.%X0 = true AND #IN_SW.%X1 = true) OR
	  (#IN_SW.%X2 = true AND #IN_SW.%X3 = false AND #IN_SW.%X4 = false AND #IN_SW.%X6 = false AND #IN_SW.%X7 = false);
	
	  //Enable PLC Control
	  #Q_CW.%X0 := false;
	  #Q_CW.%X1 := false;
	  #Q_CW.%X2 := true;
	  #Q_CW.%X3 := true;
	  #Q_CW.%X4 := #QCMD_ON = true;   // quick stop
	  #Q_CW.%X5 := true;
	  #Q_CW.%X6 := (#QCMD_ON = true AND #Drive_OK = true);
	  #Q_CW.%X7 := #OP_RESET;
	  #Q_CW.%X8 := false;
	  #Q_CW.%X9 := false;
	  #Q_CW.%X10 := true;
	  #Q_CW.%X11 := false;
	  #Q_CW.%X12 := false;
	  #Q_CW.%X13 := false;
	  #Q_CW.%X14 := false;
	  #Q_CW.%X15 := false;
	  //Drive ON/OFF
	 // IF #QCMD_ON = true THEN
	 //     #Q_CW.%X6 := true;
	 // ELSIF #QCMD_ON = FALSE THEN
	 //     #Q_CW.%X6 := FALSE;
	 // END_IF;
	  //Drive Reversing
	  //IF #drive_reversing = true THEN
	 // #Q_CW.%X11 := true;
	 // ELSIF  #drive_reversing = FALSE THEN
	 //   #Q_CW.%X11 := FALSE;
	 // END_IF;
	//Drive Fault Reset
	 // IF #OP_RESET = true THEN
	 //     #Q_CW.%X7 := true;
	 // ELSIF #OP_RESET = FALSE THEN
	 //     #Q_CW.%X7 := FALSE;
	 // END_IF;
	  (*******************************************************************
	    Network 10: Feedbacks for Running monitoring in process and simulation mode
	  ********************************************************************)
	  IF #QSIM=false AND #QMON=true  THEN
	  // Feedback monitoring in process mode
	    #TSTARTING(IN:=#QSTARTING,
	               PT:=#MON_T,
	               Q=>#MON_ERR_STARTING,
	               ET=>#QMON_T);
	     
	    #TSTOPPING(IN:=#QSTOPPING,
	              PT:=#MON_T_STOP,
	              Q=>#MON_ERR_STOPPING,
	              ET=>#QMON_T_STOP);
	    // Feedback error
	   #FB_ERR := (#QRUN AND NOT #QFB_RUN) OR (#QSTOP AND #QFB_RUN);
	    IF #FB_ERR=true OR #MON_ERR_STARTING=true OR #MON_ERR_STOPPING=true THEN
	      #QMON_ERR:=true;
	    END_IF;
	    
	    
	  ELSIF #QSIM=true AND #QMON=true THEN
	    // Feedback monitoring in simulation mode
	    #TSTARTING_SIM(IN:=#QSTARTING,
	                  PT:=#SIM_T,
	                  Q=>#MON_SIM_STARTING,
	                  ET=>#QSIM_T);
	    
	    #TSTOPPING_SIM(IN:=#QSTOPPING,
	                  PT:=#SIM_T_STOP,
	                  Q=>#MON_SIM_STOPPING,
	                  ET=>#QSIM_T_STOP);
	    
	    // Feedback for start/stop motor in simulation mode
	    IF #MON_SIM_STOPPING=true OR #QERR=true THEN
	      // Feedback for stop
	      #FB_SIM:=false;
	    ELSIF #MON_SIM_STARTING=true THEN
	      // Feedback for start
	      #FB_SIM:=true;
	    END_IF;
	  END_IF;
	
	  (*******************************************************************
	    Network 11: Feedbacks for flow monitoring in process and simulation mode
	  ********************************************************************)
	// Delay time for feedbak flow monitoring
	  #START_FLOW_TIME:=#QFLOW_MON AND (#QSTARTING OR #QRUN) AND NOT #QFLOW_MON_ACK;
	  #TFLOW(IN:=#START_FLOW_TIME,
	         PT:=#FLOW_MT,
	         Q=>#MON_ERR_FLOW,
	         ET=>#QFLOW_MT);
	  
	  //
	  #START_FLOW_TIME2:=false;
	  IF (#FLOW < #FLOW_LL) THEN
	    #START_FLOW_TIME2:=true;
	  END_IF;
	  
	     #TFLOW(IN:=#START_FLOW_TIME2,
	         PT:=#FLOW_MT,
	         Q=>#MON_ERR_FLOW2,
	         ET=>#QFLOW_MT);
	   IF #MON_ERR_FLOW2 THEN
	      #QFLOW_ERR:=true;
	   END_IF;
	  (**********************************************
	    Network 12: Drive Set Speed
	   ***********************************************)
	   //Drive Setpoint Speed in Hz
	   #SP_SpeedHz := #IN_SP_Speed / 2;
	   //Limit Speed 0 to 50 Hz
	   IF #SP_SpeedHz<0.0 THEN
	       GOTO N004;
	   END_IF;
	   IF #SP_SpeedHz > 50.0 THEN
	        GOTO N004;
	    END_IF;
	//OUT = [ ((IN–LO_LIM)/(HI_LIM–LO_LIM)) ∗ (K2–K1) ] + K1
	//UNSCALE Setpoint Speed VSD with hardwire
	//#Q_SP := REAL_TO_INT(((((#IN_SP / 2) - #SP_Lo) / (#SP_Hi - #SP_Lo)) * (#SP_K2 - #SP_K1)) + #SP_K1);
	    IF #FB_MODE = TRUE THEN
	        #Q_SP_Speed := DINT_TO_WORD(ROUND(#SP_SpeedHz * real#100.0) * DINT#27648 / DINT#5000);
	        #Drive_Actual_Speed := (INT_TO_REAL(#"IN _AV") / 27648.0 * 100.0);
	    ELSIF #FB_MODE = FALSE THEN
	        #Q_SP_Speed := DINT_TO_WORD(ROUND(#SP_SpeedHz * real#100.0) * DINT#16384 / DINT#5000);
	        #Drive_Actual_Speed := (INT_TO_REAL(#"IN _AV") / 16354.0 * 100.0);
	    END_IF;
	N004:  ;
	    
	   (**********************************************
	    Network 13: Drive Actual
	  ***********************************************)
	    #QAct_Speed := #Drive_Actual_Speed;
	 //   #QAct_Volt := (INT_TO_REAL(#IN_Volt) / 16354.0 * 1000.0);
	//    #QAct_Amp := (INT_TO_REAL(#IN_Ampere) / 16354.0 * 100.0);
	//    #QAct_KW := (INT_TO_REAL(#IN_KW) / 16354.0 * 100.0);
	//    #QAct_Nm := (INT_TO_REAL(#IN_Nm) / 16354.0 * 100.0);
	
	  (**********************************************
	    Network 14: Check errors
	  ***********************************************)
	   //Drive Fault
	   #QDrive_Fault := #IN_SW.%X3;
	   //Drive Alarm
	   #QDrive_Alarm := #IN_SW.%X7;
	   // External error
	  #QERR_EXT:=#ERR_EXTERN;  
	  // Interlock error
	  IF #LOCK=true AND ( #QSTARTING=true OR #QRUN=true) THEN
	    #QLOCK:=true;
	  END_IF;
	  //
	  IF #MPS=true THEN
	    #QMPS:=true;
	  END_IF;
	  
	  // Error in valve condition
	  #CON_ERR:=NOT((#QSTOP AND NOT #QSTARTING AND NOT #QRUN AND NOT #QSTOPPING) OR
	  (NOT #QSTOP AND #QSTARTING AND NOT #QRUN AND NOT #QSTOPPING) OR
	  (NOT #QSTOP AND NOT #QSTARTING AND #QRUN AND NOT #QSTOPPING) OR
	  (NOT #QSTOP AND NOT #QSTARTING AND NOT #QRUN AND #QSTOPPING));
	
	  (**********************************************
	    Network 15: General error
	  ***********************************************)
	  #QERR:=#QDrive_Fault OR #QDrive_Alarm OR #QERR_EXT OR #QMON_ERR OR #QFLOW_ERR OR #QMPS OR #QLOCK OR #CON_ERR;
	  
	  (**********************************************
	    Network 16: If error then stop
	  ***********************************************)
	  IF #QERR=true THEN
	    #QSTOP:=true;
	    #QSTARTING:=false;
	    #QRUN:=false;
	    #QSTOPPING:=false;
	    #QwState:=0;
	  END_IF;
	  // Reset errors
	  IF #OP_RESET=true THEN
	    #QMON_ERR:=false;
	    #QLOCK:=false;
	    #QFLOW_ERR:=false;
	    #QMPS:=false;
	  END_IF;
	    // End normal case
	END_IF;
	
	(****************************************************
	  Network 13: Influence visibility of faceplate window
	*****************************************************)
	IF #OP_VISIBILITY<>#VISIBILITY_OLD THEN
	  #VISIBILITY_OLD:=#OP_VISIBILITY;
	  #VISIBILITY:=#OP_VISIBILITY;
	ELSIF #VISIBILITY<>#VISIBILITY_OLD THEN
	  #VISIBILITY_OLD:=#VISIBILITY;
	  #OP_VISIBILITY:=#VISIBILITY;
	END_IF;
	(********************************
	  Network 14: Set state for HMI
	*********************************)
	#QdwState.%X0:=#QSTOP AND NOT #QERR;
	#QdwState.%X1:=#QSTARTING;
	#QdwState.%X2:=#QRUN;
	#QdwState.%X3:=#QSTOPPING;
	#QdwState.%X4:=false;
	#QdwState.%X5:=false;
	#QdwState.%X6:=false;
	#QdwState.%X7:=false;
	#QdwState.%X8:=#QMON;
	#QdwState.%X9:=#QMON_ERR;
	#QdwState.%X10:=#QFLOW_MON;
	#QdwState.%X11:=#QFLOW_ERR;
	#QdwState.%X12:=#QMPS;
	#QdwState.%X13:=#QDrive_Fault;
	#QdwState.%X14:=#QDrive_Alarm;
	#QdwState.%X15:=false;
	#QdwState.%X16:=#QMAN_AUT;
	#QdwState.%X17:=#QREMOTE;
	#QdwState.%X18:=#QSIM;
	#QdwState.%X19:=false;
	#QdwState.%X20:=false;
	#QdwState.%X21:=false;
	#QdwState.%X22:=false;
	#QdwState.%X23:=false;
	#QdwState.%X24:=#QERR;
	#QdwState.%X25:=#QERR_EXT;
	#QdwState.%X26:=#QLOCK;
	#QdwState.%X27:=#LOCK;
	#QdwState.%X28:=false;
	#QdwState.%X29:=false;
	#QdwState.%X30:=false;
	#QdwState.%X31:=false;
	
	(********************************
	  Network 15: Bit alarm procedure
	*********************************)
	#QwAlarm.%X0:=#QMON_ERR;
	#QwAlarm.%X1:=#QFLOW_ERR;
	#QwAlarm.%X2:=#MPS;
	#QwAlarm.%X3:=#QDrive_Fault;
	#QwAlarm.%X4:=#QLOCK;
	#QwAlarm.%X5:=#QDrive_Alarm;
	#QwAlarm.%X6:=#QERR_EXT;
	#QwAlarm.%X7:=#QERR;
	#QwAlarm.%X8:=#QSTOP;
	#QwAlarm.%X9:=#QSTARTING;
	#QwAlarm.%X10:=#QRUN;
	#QwAlarm.%X11:=#QSTOPPING;
	#QwAlarm.%X12:=#LOCK;
	#QwAlarm.%X13:=#QREMOTE;
	#QwAlarm.%X14:=#QMAN_AUT;
	#QwAlarm.%X15:=#QSIM;
END_FUNCTION_BLOCK

FUNCTION_BLOCK "Motor"
TITLE = Motor
{ S7_Optimized_Access := 'FALSE' }
AUTHOR : RM
VERSION : 0.1
//Interface FB for a motor
   VAR_INPUT 
      LOCK : Bool;   // 1 = Interlock active
      ERR_EXTERN : Bool;   // 1 = External error arised
      LIOP_SEL : Bool;   // 0 = Operator; 1 = Linking
      L_AUT : Bool;   // 0 = Manual; 1 = Automatic
      L_REMOTE : Bool;   // 0 = Local; 1 = Remote
      L_SIM : Bool;   // 0 = Normal; 1 = Simulation
      L_RESET : Bool;   // 1 = Reset error peripherie
      AUT_ON : Bool;   // 1 = CMD ON Automatic
      MAN_ON : Bool;   // 1 = CMD ON Manual
      SIM_ON : Bool;   // 1 = CMD ON Simulation
      FB_ON : Bool;   // 1 = Feedback Motor ON
      L_MON : Bool;   // 1 = Monitoring ON
      MON_T : Time := t#5s;   // Monitoring starting time in process mode
      MON_T_STOP : Time := t#5s;   // Monitoring stopping time in process mode
      MPS : Bool;   // 1 = Motor protection switch ON
      L_FLOW_MON : Bool;   // 1 = Monitoring flow
      FLOW : Real;   // Current flow
      FLOW_LL : Real := 5.0;   // Low level flow
      FLOW_MT : Time := t#8s;   // Delay of monitoring lower flow
      INSTANCE : String := 'Motor_001';   // Filter attribute for message view, also used for labelling
      RESTART : Bool;   // 1 = Initialize FB at startup (first cycle of PLC)
   END_VAR

   VAR_OUTPUT 
      QdwState : DWord;   // Status HMI
      QwState : Int;   // Motor: 0 = Stop; 1 = Starting; 2 = Run; 3 = Stopping
      QSTOPPING : Bool;   // 1 = Stopping
      QSTOP : Bool;   // 1 = Stop
      QSTARTING : Bool;   // 1 = Starting
      QRUN : Bool;   // 1 = Run
      QCMD_ON : Bool;   // 0 = Stop; 1 = Start (automatic & manual mode)
      QMON : Bool;   // 1 = Monitoring is ON
      QMON_ERR : Bool;   // 1 = Monitoring errror
      QMON_T : Time;   // Expierd starting time in process mode
      QMON_T_STOP : Time;   // Expierd stopping time in process mode
      QFLOW_MON : Bool;   // 1 = Flow monitoring is ON
      QFLOW_MT : Time;   // Expiered delay of monitoring lower flow
      QFLOW_ERR : Bool;   // 1 = Error flow monitoring
      QMPS : Bool;   // 1 = Motor protecting switch
      QMAN_AUT : Bool;   // 0 = Manual; 1 = Automatic
      QREMOTE : Bool;   // 0 = Local; 1 = Remote
      QSIM : Bool;   // 0 = Normal; 1 = Simulation
      QLOCK : Bool;   // 1 = Interlock is active
      QERR : Bool;   // 1 = Common error
      QERR_EXT : Bool;   // 1 = External error
      QwAlarm : Word;   // Bit alarm procedure
   END_VAR

   VAR_IN_OUT 
      VISIBILITY : Byte;   // Bit 0: Tab1 of window; Bit 1: Tab2 of window; ... ; Bit 7: Minimize
      OPdwCmd : DWord;   // Contorl word HMI
   END_VAR

   VAR 
      FB_SIM : Bool;
      SIM_T : Time;
      QSIM_T : Time;
      SIM_T_STOP : Time;
      QSIM_T_STOP : Time;
      QCMD_SIM : Bool;
      OP_RESET : Bool;   // Reset errors
      QFLOW_MON_ACK : Bool;
      OP_VISIBILITY : Byte;   // Bit 0: Tab1 of window; Bit 1: Tab2 of window; ... ; Bit 7: Minimize
      VISIBILITY_OLD : Byte;   // Save last status of VISIBILITY
      SE_L_RESET_LINK : Bool;   // Signal edge for the reset input from linking
      SE_L_RESET_LINK_COND : Bool;   // Condition of signal edge
      SE_L_RESET_OP : Bool;   // Signal edge for the reset input from operator
      TSTARTING {InstructionName := 'TON_TIME'; LibVersion := '1.0'} : TON_TIME;
      TSTOPPING {InstructionName := 'TON_TIME'; LibVersion := '1.0'} : TON_TIME;
      TFLOW {InstructionName := 'TON_TIME'; LibVersion := '1.0'} : TON_TIME;
      TSTARTING_SIM {InstructionName := 'TON_TIME'; LibVersion := '1.0'} : TON_TIME;
      TSTOPPING_SIM {InstructionName := 'TON_TIME'; LibVersion := '1.0'} : TON_TIME;
   END_VAR

   VAR_TEMP 
      CON_ERR : Bool;   // Error in motor condition
      MON_ERR_STARTING : Bool;   // Monitoring error for starting motor in process mode
      MON_ERR_STOPPING : Bool;   // Monitoring error for stopping motor in process mode
      MON_SIM_STARTING : Bool;   // Monitoring error for starting motor in simulation mode
      MON_SIM_STOPPING : Bool;   // Monitoring error for stopping motor in simulation mode
      FB_ERR : Bool;   // Feedback error in process mode
      MON_ERR_FLOW2 : Bool;
      START_FLOW_TIME2 : Bool;
      START_FLOW_TIME : Bool;   // Start Signal of delay time for flow
      MON_ERR_FLOW : Bool;   // Monitoring error for flow
   END_VAR


BEGIN
	(********************************
	           Start up
	*********************************)
	IF #RESTART= true THEN
	  // Restart case
	  #QCMD_ON:= false;
	  #QSTOP:=true;
	  #QSTOPPING:=false;
	  #QRUN:=false;
	  #QSTARTING:=false;
	  #VISIBILITY:=0;
	  #OPdwCmd:=0;
	ELSE
	  // Normal case
	  
	  (******************************************
	    Network 1: Operating mode: manual/automatic
	    Vaiable: OPdwCmd  Bit:  16  =  Manual
	    Vaiable: OPdwCmd  Bit:  17  =  Automatic
	  *******************************************)
	  IF (#LIOP_SEL=true AND #L_AUT=true) OR (#OPdwCmd.%X17=true AND #LIOP_SEL=false) THEN
	    #QMAN_AUT:=true;
	    #OPdwCmd.%X16:=false;
	    #OPdwCmd.%X17:=false;
	  ELSIF (#LIOP_SEL=true AND #L_AUT=false) OR (#OPdwCmd.%X16=true AND #LIOP_SEL=false) THEN
	    #QMAN_AUT:= false;
	    #OPdwCmd.%X16:=false;
	    #OPdwCmd.%X17:=false;
	  END_IF;
	  
	  (******************************************
	    Network 2: Control mode: local/remote
	    Vaiable: OPdwCmd  Bit:  18  =  Local
	    Vaiable: OPdwCmd  Bit:  19  =  Remote
	  *******************************************)
	  IF (#LIOP_SEL=true AND #L_REMOTE=true) OR (#OPdwCmd.%X19=true AND #LIOP_SEL=false) THEN
	    #QREMOTE:=true;
	    #OPdwCmd.%X18:=false;
	    #OPdwCmd.%X19:=false;
	  ELSIF (#LIOP_SEL=true AND #L_REMOTE=false) OR (#OPdwCmd.%X18=true AND #LIOP_SEL=false) THEN
	    #QREMOTE:= false;
	    #OPdwCmd.%X18:=false;
	    #OPdwCmd.%X19:=false;
	  END_IF;
	  
	  (******************************************
	    Network 3: Simulation On/Off
	    Vaiable: OPdwCmd  Bit:  20  =  Process
	    Vaiable: OPdwCmd  Bit:  21  =  Simulation
	  *******************************************)
	  IF (#LIOP_SEL=true AND #L_SIM=true) OR (#OPdwCmd.%X21=true AND #LIOP_SEL=false) THEN
	    #QSIM:=true;
	    #OPdwCmd.%X20:=false;
	    #OPdwCmd.%X21:=false;
	  ELSIF (#LIOP_SEL=true AND #L_SIM=false) OR (#OPdwCmd.%X20=true AND #LIOP_SEL=false) THEN
	    #QSIM:= false;
	    #OPdwCmd.%X20:=false;
	    #OPdwCmd.%X21:=false;
	  END_IF;
	  
	  (*************************************
	    Network 4: Reset Operation
	    Vaiable: OPdwCmd  Bit:  24  =  Reset
	  **************************************)
	  // Rising edge by linking
	  IF #L_RESET=true AND #SE_L_RESET_LINK_COND=false THEN
	    #SE_L_RESET_LINK:=true;
	    #SE_L_RESET_LINK_COND:=true;
	  ELSIF #L_RESET=true AND #SE_L_RESET_LINK_COND=true THEN
	    #SE_L_RESET_LINK:=false;
	  ELSE
	    #SE_L_RESET_LINK_COND:=false;
	  END_IF;
	  // Rising edge by operator
	  IF #OPdwCmd.%X24=true THEN
	    #SE_L_RESET_OP:=true;
	    #OPdwCmd.%X24:=false;
	  ELSE
	    #SE_L_RESET_OP:=false;
	  END_IF;
	  // Reset error
	  #OP_RESET:=(#L_RESET) OR (#SE_L_RESET_OP AND NOT #LIOP_SEL) AND NOT #LOCK;
	  
	  (**********************************************
	    Network 5: Monitoring feedback ON/OFF
	    Vaiable: OPdwCmd  Bit:  8  =  Monitoring ON
	    Vaiable: OPdwCmd  Bit:  9  =  Monitoring OFF
	  ***********************************************)
	  IF (#LIOP_SEL=true AND #L_MON=false) OR (#OPdwCmd.%X9=true AND #LIOP_SEL=false)THEN
	    #QMON:=false;
	    #OPdwCmd.%X8:=false;
	    #OPdwCmd.%X9:=false;
	  ELSIF (#LIOP_SEL=true AND #L_MON=true) OR (#OPdwCmd.%X8=true AND #LIOP_SEL=false)THEN
	    #QMON:=true;
	    #OPdwCmd.%X8:=false;
	    #OPdwCmd.%X9:=false;
	  END_IF;
	  
	  (***************************************************
	    Network 6: Monitoring flow ON/OFF
	    Vaiable: OPdwCmd  Bit:  10  =  Monitoring flow ON
	    Vaiable: OPdwCmd  Bit:  11  =  Monitoring flow OFF
	  ****************************************************)
	  IF (#LIOP_SEL=true AND #L_FLOW_MON=false) OR (#OPdwCmd.%X11=true AND #LIOP_SEL=false)THEN
	    #QFLOW_MON:=false;
	    #OPdwCmd.%X10:=false;
	    #OPdwCmd.%X11:=false;
	  ELSIF (#LIOP_SEL=true AND #L_FLOW_MON=true) OR (#OPdwCmd.%X10=true AND #LIOP_SEL=false)THEN
	    #QFLOW_MON:=true;
	    #OPdwCmd.%X10:=false;
	    #OPdwCmd.%X11:=false;
	  END_IF;
	  
	   (**********************************************
	    Network 6: START/STOP Motor
	    Vaiable: OPdwCmd  Bit:  0  =  STOP Motor
	    Vaiable: OPdwCmd  Bit:  1  =  START Motor
	  ***********************************************)
	  IF #QERR=false THEN
	    // No errors occurs
	    IF #QSIM=false THEN
	     // Simulation mode is not active
	      // Automatic/Manual mode
	      IF #QMAN_AUT=true THEN
	        // Automatic mode is active
	        // OPEN/CLOSE valve by linking (AUT_ON)
	        #QCMD_ON:=#AUT_ON;
	        #OPdwCmd.%X0:=false;
	        #OPdwCmd.%X1:=false;
	      ELSE
	       // Automatic mode is not active
	        // Local/Remote mode
	        IF #QREMOTE=false THEN
	          // Local mode is active
	          // OPEN/CLOSE valve by linking (MAN_ON)
	          #QCMD_ON:=#MAN_ON AND NOT #QMAN_AUT;
	          #OPdwCmd.%X0:=false;
	          #OPdwCmd.%X1:=false;
	        ELSE
	         // Remote mode is active
	          // Open valve by operator
	          IF #OPdwCmd.%X1=true THEN
	            #QCMD_ON:=true;
	            #OPdwCmd.%X0:=false;
	            #OPdwCmd.%X1:=false;
	          END_IF;
	          // Close valve by operator
	          IF #OPdwCmd.%X0=true THEN
	            #QCMD_ON:=false;
	            #OPdwCmd.%X0:=false;
	            #OPdwCmd.%X1:=false;
	          END_IF;
	        END_IF;
	      END_IF;
	    ELSE
	      // Local/Remote mode
	      IF #QREMOTE=false THEN
	        // Local mode is active
	          // OPEN/CLOSE valve by linking (SIM_ON)
	          #QCMD_SIM:=#SIM_ON;
	          #OPdwCmd.%X0:=false;
	          #OPdwCmd.%X1:=false;
	      ELSE
	        // Remote mode is active
	          // Open valve by operator
	          IF #OPdwCmd.%X1=true THEN
	            #QCMD_SIM:=true;
	            #OPdwCmd.%X0:=false;
	            #OPdwCmd.%X1:=false;
	          END_IF;
	          // Close valve by operator
	          IF #OPdwCmd.%X0=true THEN
	            #QCMD_SIM:=false;
	            #OPdwCmd.%X0:=false;
	            #OPdwCmd.%X1:=false;
	          END_IF;        
	       END_IF;
	    END_IF;  
	  ELSE
	    // Errors occurs
	    #QCMD_ON:=false;
	    #QCMD_SIM:=false;
	    #OPdwCmd.%X0:=false;
	    #OPdwCmd.%X1:=false;
	  END_IF;
	  
	  (****************************************
	    Network 7: Control signal to the valve
	  *****************************************)
	  IF #QERR=false THEN
	    // Motor is stopped
	    IF (((#FB_ON=false OR #QMON=false) AND #QSIM=false AND #QCMD_ON=false) OR
	      ((#FB_SIM=false OR #QMON=false) AND #QSIM=true AND #QCMD_SIM=false)) AND #QSTOPPING=true THEN
	      #QSTOP:=true;
	      #QSTOPPING:=false;
	      #QRUN:=false;
	      #QSTARTING:=false;
	      #QwState:=0;
	    END_IF;
	    // Motor is stopping
	    IF ((#QSIM=false AND #QCMD_ON=false) OR (#QSIM=true AND #QCMD_SIM=false)) AND (#QRUN=true OR #QSTARTING=true) THEN
	      #QSTOP:=false;
	      #QSTOPPING:=true;
	      #QRUN:=false;
	      #QSTARTING:=false;
	      #QwState:=3;
	    END_IF;
	    // Motor is running 
	    IF (((#FB_ON=true OR #QMON=false) AND #QSIM=false AND #QCMD_ON=true) OR
	      ((#FB_SIM=true OR #QMON=false) AND #QSIM=true AND #QCMD_SIM=true)) AND #QSTARTING=true THEN    
	    #QSTOP:=false;
	    #QSTOPPING:=false;
	    #QRUN:=true;
	    #QSTARTING:=false;
	    #QwState:=2;
	    END_IF;
	    // Motor is starting 
	    IF ((#QSIM=false AND #QCMD_ON=true) OR (#QSIM=true AND #QCMD_SIM=true)) AND #QSTOP=true THEN
	    #QSTOP:=false;
	    #QSTOPPING:=false;
	    #QRUN:=false;
	    #QSTARTING:=true;
	    #QwState:=1;
	    END_IF;
	  END_IF;
	  
	  (*******************************************************************
	    Network 8: Feedbacks for monitoring in process and simulation mode
	  ********************************************************************)
	  IF #QSIM=false AND #QMON=true  THEN
	  // Feedback monitoring in process mode
	    #TSTARTING(IN:=#QSTARTING,
	               PT:=#MON_T,
	               Q=>#MON_ERR_STARTING,
	               ET=>#QMON_T);
	     
	    #TSTOPPING(IN:=#QSTOPPING,
	              PT:=#MON_T_STOP,
	              Q=>#MON_ERR_STOPPING,
	              ET=>#QMON_T_STOP);
	    // Feedback error
	    #FB_ERR:= (#QRUN AND NOT #FB_ON) OR (#QSTOP AND #FB_ON);
	    IF #FB_ERR=true OR #MON_ERR_STARTING=true OR #MON_ERR_STOPPING=true THEN
	      #QMON_ERR:=true;
	    END_IF;
	    
	    
	  ELSIF #QSIM=true AND #QMON=true THEN
	    // Feedback monitoring in simulation mode
	    #TSTARTING_SIM(IN:=#QSTARTING,
	                  PT:=#SIM_T,
	                  Q=>#MON_SIM_STARTING,
	                  ET=>#QSIM_T);
	    
	    #TSTOPPING_SIM(IN:=#QSTOPPING,
	                  PT:=#SIM_T_STOP,
	                  Q=>#MON_SIM_STOPPING,
	                  ET=>#QSIM_T_STOP);
	    
	    // Feedback for start/stop motor in simulation mode
	    IF #MON_SIM_STOPPING=true OR #QERR=true THEN
	      // Feedback for stop
	      #FB_SIM:=false;
	    ELSIF #MON_SIM_STARTING=true THEN
	      // Feedback for start
	      #FB_SIM:=true;
	    END_IF;
	  END_IF;
	
	  (*******************************************************************
	    Network 9: Feedbacks for flow monitoring in process and simulation mode
	  ********************************************************************)
	// Delay time for feedbak flow monitoring
	  #START_FLOW_TIME:=#QFLOW_MON AND (#QSTARTING OR #QRUN) AND NOT #QFLOW_MON_ACK;
	  #TFLOW(IN:=#START_FLOW_TIME,
	         PT:=#FLOW_MT,
	         Q=>#MON_ERR_FLOW,
	         ET=>#QFLOW_MT);
	  
	  //
	  #START_FLOW_TIME2:=false;
	  IF (#FLOW < #FLOW_LL) THEN
	    #START_FLOW_TIME2:=true;
	  END_IF;
	  
	     #TFLOW(IN:=#START_FLOW_TIME2,
	         PT:=#FLOW_MT,
	         Q=>#MON_ERR_FLOW2,
	         ET=>#QFLOW_MT);
	IF #MON_ERR_FLOW2 THEN
	  #QFLOW_ERR:=true;
	END_IF;
	
	  (**********************************************
	    Network 10: Check errors
	  ***********************************************)
	  // External error
	  #QERR_EXT:=#ERR_EXTERN;  
	  // Interlock error
	  IF #LOCK=true AND ( #QSTARTING=true OR #QRUN=true) THEN
	    #QLOCK:=true;
	  END_IF;
	  //
	  IF #MPS=true THEN
	    #QMPS:=true;
	  END_IF;
	  
	  // Error in valve condition
	  #CON_ERR:=NOT((#QSTOP AND NOT #QSTARTING AND NOT #QRUN AND NOT #QSTOPPING) OR
	  (NOT #QSTOP AND #QSTARTING AND NOT #QRUN AND NOT #QSTOPPING) OR
	  (NOT #QSTOP AND NOT #QSTARTING AND #QRUN AND NOT #QSTOPPING) OR
	  (NOT #QSTOP AND NOT #QSTARTING AND NOT #QRUN AND #QSTOPPING));
	
	  (**********************************************
	    Network 11: General error
	  ***********************************************)
	  #QERR:= #QERR_EXT OR #QMON_ERR OR #QFLOW_ERR OR #QMPS OR #QLOCK OR #CON_ERR;
	  
	  (**********************************************
	    Network 12: If error then stop
	  ***********************************************)
	  IF #QERR=true THEN
	    #QSTOP:=true;
	    #QSTARTING:=false;
	    #QRUN:=false;
	    #QSTOPPING:=false;
	    #QwState:=0;
	  END_IF;
	  // Reset errors
	  IF #OP_RESET=true THEN
	    #QMON_ERR:=false;
	    #QLOCK:=false;
	    #QFLOW_ERR:=false;
	    #QMPS:=false;
	  END_IF;
	    // End normal case
	END_IF;
	
	(****************************************************
	  Network 13: Influence visibility of faceplate window
	*****************************************************)
	IF #OP_VISIBILITY<>#VISIBILITY_OLD THEN
	  #VISIBILITY_OLD:=#OP_VISIBILITY;
	  #VISIBILITY:=#OP_VISIBILITY;
	ELSIF #VISIBILITY<>#VISIBILITY_OLD THEN
	  #VISIBILITY_OLD:=#VISIBILITY;
	  #OP_VISIBILITY:=#VISIBILITY;
	END_IF;
	(********************************
	  Network 14: Set state for HMI
	*********************************)
	#QdwState.%X0:=#QSTOP AND NOT #QERR;
	#QdwState.%X1:=#QSTARTING;
	#QdwState.%X2:=#QRUN;
	#QdwState.%X3:=#QSTOPPING;
	#QdwState.%X4:=false;
	#QdwState.%X5:=false;
	#QdwState.%X6:=false;
	#QdwState.%X7:=false;
	#QdwState.%X8:=#QMON;
	#QdwState.%X9:=#QMON_ERR;
	#QdwState.%X10:=#QFLOW_MON;
	#QdwState.%X11:=#QFLOW_ERR;
	#QdwState.%X12:=#QMPS;
	#QdwState.%X13:=false;
	#QdwState.%X14:=false;
	#QdwState.%X15:=false;
	#QdwState.%X16:=#QMAN_AUT;
	#QdwState.%X17:=#QREMOTE;
	#QdwState.%X18:=#QSIM;
	#QdwState.%X19:=false;
	#QdwState.%X20:=false;
	#QdwState.%X21:=false;
	#QdwState.%X22:=false;
	#QdwState.%X23:=false;
	#QdwState.%X24:=#QERR;
	#QdwState.%X25:=#QERR_EXT;
	#QdwState.%X26:=#QLOCK;
	#QdwState.%X27:=#LOCK;
	#QdwState.%X28:=false;
	#QdwState.%X29:=false;
	#QdwState.%X30:=false;
	#QdwState.%X31:=false;
	
	(********************************
	  Network 15: Bit alarm procedure
	*********************************)
	#QwAlarm.%X0:=#QMON_ERR;
	#QwAlarm.%X1:=#QFLOW_ERR;
	#QwAlarm.%X2:=#MPS;
	#QwAlarm.%X3:=false;
	#QwAlarm.%X4:=#QLOCK;
	#QwAlarm.%X5:=false;
	#QwAlarm.%X6:=#QERR_EXT;
	#QwAlarm.%X7:=#QERR;
	#QwAlarm.%X8:=#QSTOP;
	#QwAlarm.%X9:=#QSTARTING;
	#QwAlarm.%X10:=#QRUN;
	#QwAlarm.%X11:=#QSTOPPING;
	#QwAlarm.%X12:=#LOCK;
	#QwAlarm.%X13:=#QREMOTE;
	#QwAlarm.%X14:=#QMAN_AUT;
	#QwAlarm.%X15:=#QSIM;
END_FUNCTION_BLOCK

FUNCTION "Preparation_Area" : Void   // FC12, LAD
{ S7_Optimized_Access := 'TRUE' }
VERSION : 0.1
// stored: AutoNumber false, IsIECCheckEnabled false, SetENOAutomatically false, UDAEnableTagReadback false
   VAR_TEMP   // added for the SCL form of the ladder/FBD networks
      _w1 : Bool;
      _w2 : Bool;
      _w3 : Bool;
   END_VAR
BEGIN

REGION Network 2: Analog IO
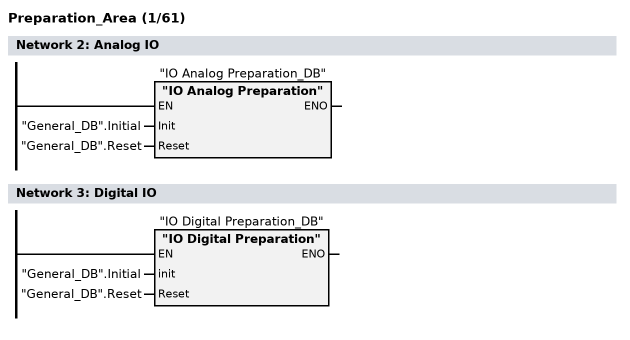
   RUNG wire#powerrail
      "IO Analog Preparation_DB"(Init := "General_DB".Initial, Reset := "General_DB".Reset)
   END_RUNG
   // the same network as SCL:
   "IO Analog Preparation_DB"(Init := "General_DB".Initial, Reset := "General_DB".Reset);   // "IO Analog Preparation"
END_REGION

REGION Network 3: Digital IO
   RUNG wire#powerrail
      "IO Digital Preparation_DB"(init := "General_DB".Initial, Reset := "General_DB".Reset)
   END_RUNG
   // the same network as SCL:
   "IO Digital Preparation_DB"(init := "General_DB".Initial, Reset := "General_DB".Reset);   // "IO Digital Preparation"
END_REGION

NETWORK
TITLE = T-02.00 DOSE ON OFF
      O     "Blend to Preparation"."T-20".Raw_Material.ChiliAwetan_1.DoseRun;
      O     "Blend to Preparation"."T-21".Raw_Material.ChiliAwetan_1.DoseRun;
      O     "Blend to Preparation"."T-30".Raw_Material.ChiliAwetan_1.DoseRun;
      O     "Blend to Preparation"."T-31".Raw_Material.ChiliAwetan_1.DoseRun;
      O     "Blend to Preparation"."T-40".Raw_Material.ChiliAwetan_1.DoseRun;
      O     "Blend to Preparation"."T-41".Raw_Material.ChiliAwetan_1.DoseRun;
      =     "T-02_ChiliAwetan_1".IN_Dose_Run;

NETWORK
TITLE = T-02.00 DOSE PAUSE
      O     "Blend to Preparation"."T-20".Raw_Material.ChiliAwetan_1.DoseHeld;
      O     "Blend to Preparation"."T-21".Raw_Material.ChiliAwetan_1.DoseHeld;
      O     "Blend to Preparation"."T-30".Raw_Material.ChiliAwetan_1.DoseHeld;
      O     "Blend to Preparation"."T-31".Raw_Material.ChiliAwetan_1.DoseHeld;
      O     "Blend to Preparation"."T-40".Raw_Material.ChiliAwetan_1.DoseHeld;
      O     "Blend to Preparation"."T-41".Raw_Material.ChiliAwetan_1.DoseHeld;
      =     "T-02_ChiliAwetan_1".IN_Dose_Held;

NETWORK
TITLE = T-02.00 DOSE VALVE CMD
      O(;
      A     "Blend to Preparation"."T-20".Raw_Material.ChiliAwetan_1.DoseRun;
      A     "Blend to Preparation"."T-20".Raw_Material.ChiliAwetan_1.ValveCMD;
      );
      O(;
      A     "Blend to Preparation"."T-21".Raw_Material.ChiliAwetan_1.DoseRun;
      A     "Blend to Preparation"."T-21".Raw_Material.ChiliAwetan_1.ValveCMD;
      );
      O(;
      A     "Blend to Preparation"."T-30".Raw_Material.ChiliAwetan_1.DoseRun;
      A     "Blend to Preparation"."T-30".Raw_Material.ChiliAwetan_1.ValveCMD;
      );
      O(;
      A     "Blend to Preparation"."T-31".Raw_Material.ChiliAwetan_1.DoseRun;
      A     "Blend to Preparation"."T-31".Raw_Material.ChiliAwetan_1.ValveCMD;
      );
      O(;
      A     "Blend to Preparation"."T-40".Raw_Material.ChiliAwetan_1.DoseRun;
      A     "Blend to Preparation"."T-40".Raw_Material.ChiliAwetan_1.ValveCMD;
      );
      O(;
      A     "Blend to Preparation"."T-41".Raw_Material.ChiliAwetan_1.DoseRun;
      A     "Blend to Preparation"."T-41".Raw_Material.ChiliAwetan_1.ValveCMD;
      );
      =     "T-02_ChiliAwetan_1".IN_Dose_Valve_Cmd;


NETWORK
TITLE = T-02.00 DOSE Pump CMD
      O(;
      A     "Blend to Preparation"."T-20".Raw_Material.ChiliAwetan_1.DoseRun;
      A     "Blend to Preparation"."T-20".Raw_Material.ChiliAwetan_1.PumpCMD;
      );
      O(;
      A     "Blend to Preparation"."T-21".Raw_Material.ChiliAwetan_1.DoseRun;
      A     "Blend to Preparation"."T-21".Raw_Material.ChiliAwetan_1.PumpCMD;
      );
      O(;
      A     "Blend to Preparation"."T-30".Raw_Material.ChiliAwetan_1.DoseRun;
      A     "Blend to Preparation"."T-30".Raw_Material.ChiliAwetan_1.PumpCMD;
      );
      O(;
      A     "Blend to Preparation"."T-31".Raw_Material.ChiliAwetan_1.DoseRun;
      A     "Blend to Preparation"."T-31".Raw_Material.ChiliAwetan_1.PumpCMD;
      );
      O(;
      A     "Blend to Preparation"."T-40".Raw_Material.ChiliAwetan_1.DoseRun;
      A     "Blend to Preparation"."T-40".Raw_Material.ChiliAwetan_1.PumpCMD;
      );
      O(;
      A     "Blend to Preparation"."T-41".Raw_Material.ChiliAwetan_1.DoseRun;
      A     "Blend to Preparation"."T-41".Raw_Material.ChiliAwetan_1.PumpCMD;
      );
      =     "T-02_ChiliAwetan_1".IN_Dose_Pump_Cmd;



NETWORK
TITLE = T-02.00 DOSE PUMP SPEED
// Checking
      O     "Blend to Preparation"."T-20".Raw_Material.ChiliAwetan_1.DoseRun;
      JC    SP_02_FROM_20;
      O     "Blend to Preparation"."T-21".Raw_Material.ChiliAwetan_1.DoseRun;
      JC    SP_02_FROM_21;
      O     "Blend to Preparation"."T-30".Raw_Material.ChiliAwetan_1.DoseRun;
      JC    SP_02_FROM_30;
      O     "Blend to Preparation"."T-31".Raw_Material.ChiliAwetan_1.DoseRun;
      JC    SP_02_FROM_31;
      O     "Blend to Preparation"."T-40".Raw_Material.ChiliAwetan_1.DoseRun;
      JC    SP_02_FROM_40;
      O     "Blend to Preparation"."T-41".Raw_Material.ChiliAwetan_1.DoseRun;
      JC    SP_02_FROM_41;
//Jump to end if Blend not Dosing
      JC    SP_02_SELF;
//Load Set Point
SP_02_FROM_20:L     "Blend to Preparation".Recipe."T-20".ChiliAwetan_1.SP_PumpSpeed;
      T     "T-02_ChiliAwetan_1".IN_Dose_Pump_Sp;
      JC    SP_02_SELF;
SP_02_FROM_21:L     "Blend to Preparation".Recipe."T-21".ChiliAwetan_1.SP_PumpSpeed;
      T     "T-02_ChiliAwetan_1".IN_Dose_Pump_Sp;
      JC    SP_02_SELF;
SP_02_FROM_30:L     "Blend to Preparation".Recipe."T-30".ChiliAwetan_1.SP_PumpSpeed;
      T     "T-02_ChiliAwetan_1".IN_Dose_Pump_Sp;
      JC    SP_02_SELF;
SP_02_FROM_31:L     "Blend to Preparation".Recipe."T-31".ChiliAwetan_1.SP_PumpSpeed;
      T     "T-02_ChiliAwetan_1".IN_Dose_Pump_Sp;
      JC    SP_02_SELF;
SP_02_FROM_40:L     "Blend to Preparation".Recipe."T-40".ChiliAwetan_1.SP_PumpSpeed;
      T     "T-02_ChiliAwetan_1".IN_Dose_Pump_Sp;
      JC    SP_02_SELF;
SP_02_FROM_41:L     "Blend to Preparation".Recipe."T-41".ChiliAwetan_1.SP_PumpSpeed;
      T     "T-02_ChiliAwetan_1".IN_Dose_Pump_Sp;
      JC    SP_02_SELF;
// END
SP_02_SELF:L     "T-02_ChiliAwetan_1".IN_Dose_Pump_Sp;
      T     "T-02_ChiliAwetan_1".IN_Dose_Pump_Sp;


NETWORK
TITLE = T-02.00 Header Req
// HEADER 1 Req
      O     "Blend to Preparation"."T-20".Raw_Material.ChiliAwetan_1.Header1_Req;
      O     "Blend to Preparation"."T-21".Raw_Material.ChiliAwetan_1.Header1_Req;
      O     "Blend to Preparation"."T-30".Raw_Material.ChiliAwetan_1.Header1_Req;
      O     "Blend to Preparation"."T-31".Raw_Material.ChiliAwetan_1.Header1_Req;
      O     "Blend to Preparation"."T-40".Raw_Material.ChiliAwetan_1.Header1_Req;
      O     "Blend to Preparation"."T-41".Raw_Material.ChiliAwetan_1.Header1_Req;
      =     "T-02_ChiliAwetan_1".IN_Dose_Header_1;

// HEADER 2 Req
      O     "Blend to Preparation"."T-20".Raw_Material.ChiliAwetan_1.Header2_Req;
      O     "Blend to Preparation"."T-21".Raw_Material.ChiliAwetan_1.Header2_Req;
      O     "Blend to Preparation"."T-30".Raw_Material.ChiliAwetan_1.Header2_Req;
      O     "Blend to Preparation"."T-31".Raw_Material.ChiliAwetan_1.Header2_Req;
      O     "Blend to Preparation"."T-40".Raw_Material.ChiliAwetan_1.Header2_Req;
      O     "Blend to Preparation"."T-41".Raw_Material.ChiliAwetan_1.Header2_Req;
      =     "T-02_ChiliAwetan_1".IN_Dose_Header_2;




REGION Network 11: T-02.00 LineTransferOK
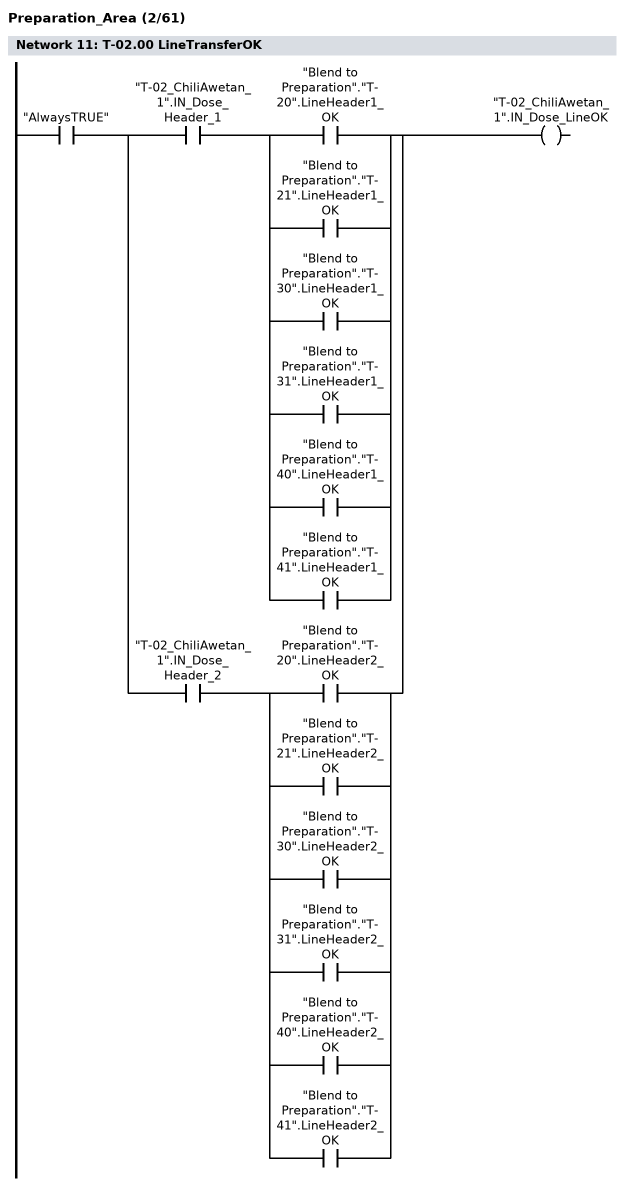
   RUNG wire#powerrail
      Contact( "AlwaysTRUE" )
      wire#w1
      Contact( "T-02_ChiliAwetan_1".IN_Dose_Header_1 )
      wire#w2
      Contact( "Blend to Preparation"."T-20".LineHeader1_OK )
      wire#w3
      Coil( "T-02_ChiliAwetan_1".IN_Dose_LineOK )
   END_RUNG
   RUNG wire#w2
      Contact( "Blend to Preparation"."T-21".LineHeader1_OK )
   END_RUNG wire#w3
   RUNG wire#w2
      Contact( "Blend to Preparation"."T-30".LineHeader1_OK )
   END_RUNG wire#w3
   RUNG wire#w2
      Contact( "Blend to Preparation"."T-31".LineHeader1_OK )
   END_RUNG wire#w3
   RUNG wire#w2
      Contact( "Blend to Preparation"."T-40".LineHeader1_OK )
   END_RUNG wire#w3
   RUNG wire#w2
      Contact( "Blend to Preparation"."T-41".LineHeader1_OK )
   END_RUNG wire#w3
   RUNG wire#w1
      Contact( "T-02_ChiliAwetan_1".IN_Dose_Header_2 )
      wire#w4
      Contact( "Blend to Preparation"."T-20".LineHeader2_OK )
   END_RUNG wire#w3
   RUNG wire#w4
      Contact( "Blend to Preparation"."T-21".LineHeader2_OK )
   END_RUNG wire#w3
   RUNG wire#w4
      Contact( "Blend to Preparation"."T-30".LineHeader2_OK )
   END_RUNG wire#w3
   RUNG wire#w4
      Contact( "Blend to Preparation"."T-31".LineHeader2_OK )
   END_RUNG wire#w3
   RUNG wire#w4
      Contact( "Blend to Preparation"."T-40".LineHeader2_OK )
   END_RUNG wire#w3
   RUNG wire#w4
      Contact( "Blend to Preparation"."T-41".LineHeader2_OK )
   END_RUNG wire#w3
   // the same network as SCL:
   "T-02_ChiliAwetan_1".IN_Dose_LineOK := "AlwaysTRUE" AND (("T-02_ChiliAwetan_1".IN_Dose_Header_1 AND ("Blend to Preparation"."T-20".LineHeader1_OK OR "Blend to Preparation"."T-21".LineHeader1_OK OR "Blend to Preparation"."T-30".LineHeader1_OK OR "Blend to Preparation"."T-31".LineHeader1_OK OR "Blend to Preparation"."T-40".LineHeader1_OK OR "Blend to Preparation"."T-41".LineHeader1_OK)) OR ("T-02_ChiliAwetan_1".IN_Dose_Header_2 AND ("Blend to Preparation"."T-20".LineHeader2_OK OR "Blend to Preparation"."T-21".LineHeader2_OK OR "Blend to Preparation"."T-30".LineHeader2_OK OR "Blend to Preparation"."T-31".LineHeader2_OK OR "Blend to Preparation"."T-40".LineHeader2_OK OR "Blend to Preparation"."T-41".LineHeader2_OK)));
END_REGION

REGION Network 12: T-02.00___Chili Awetan 1
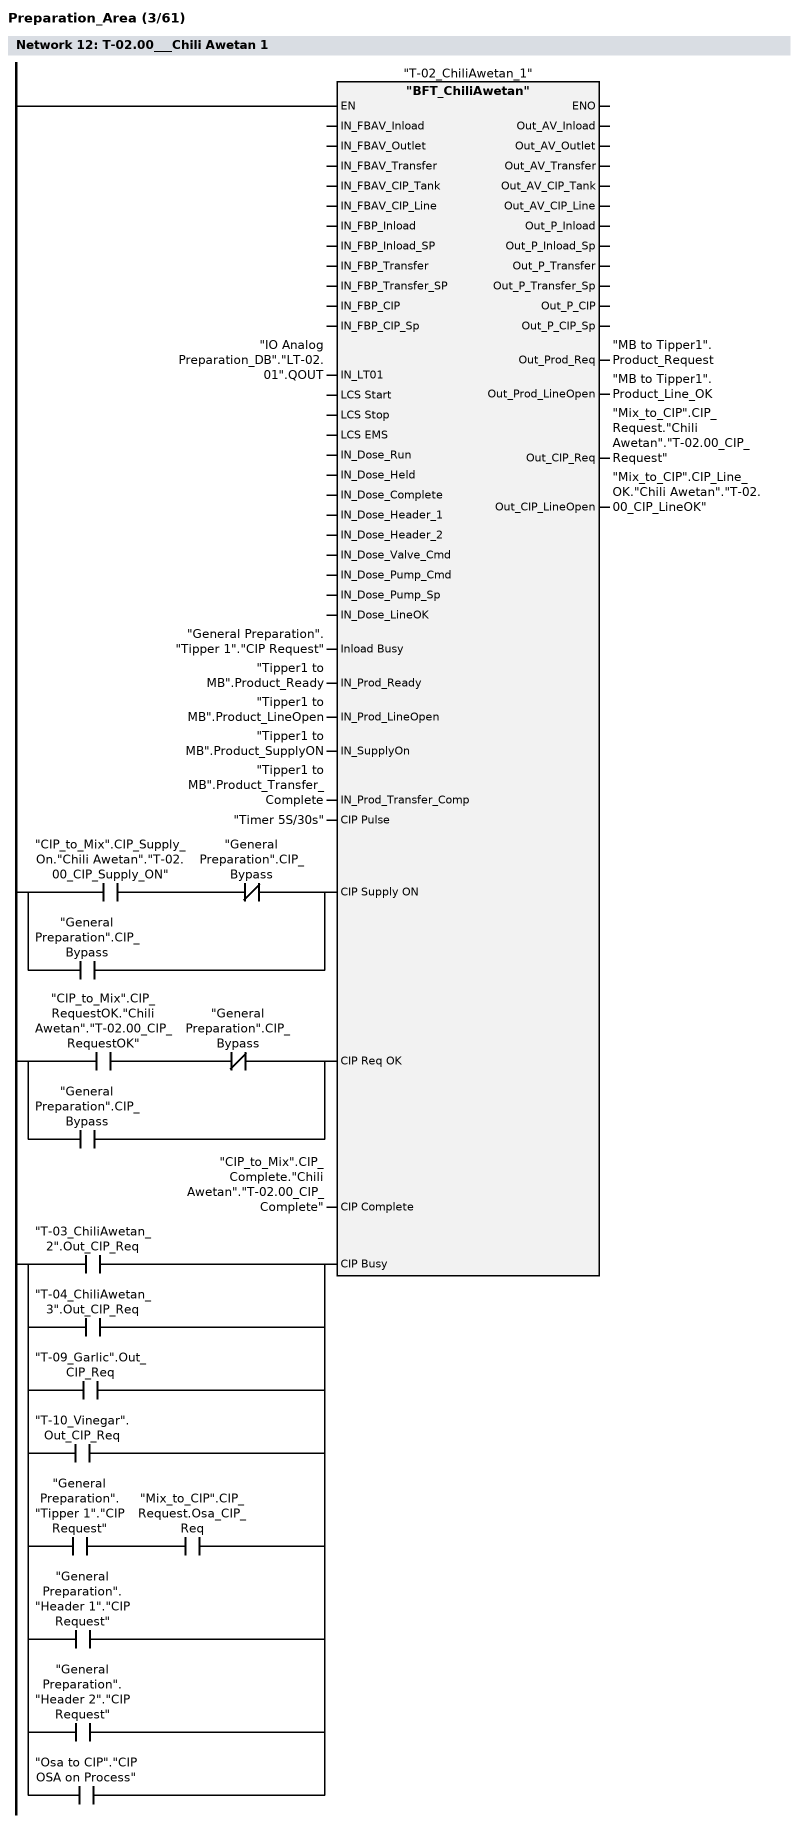
   RUNG wire#powerrail
      "T-02_ChiliAwetan_1"("CIP Supply ON" := wire#w1, "CIP Req OK" := wire#w2, "CIP Busy" := wire#w3, IN_FBAV_Inload :=, IN_FBAV_Outlet :=, IN_FBAV_Transfer :=, IN_FBAV_CIP_Tank :=, IN_FBAV_CIP_Line :=, IN_FBP_Inload :=, IN_FBP_Inload_SP :=, IN_FBP_Transfer :=, IN_FBP_Transfer_SP :=, IN_FBP_CIP :=, IN_FBP_CIP_Sp :=, IN_LT01 := "IO Analog Preparation_DB"."LT-02.01".QOUT, "LCS Start" :=, "LCS Stop" :=, "LCS EMS" :=, IN_Dose_Run :=, IN_Dose_Held :=, IN_Dose_Complete :=, IN_Dose_Header_1 :=, IN_Dose_Header_2 :=, IN_Dose_Valve_Cmd :=, IN_Dose_Pump_Cmd :=, IN_Dose_Pump_Sp :=, IN_Dose_LineOK :=, "Inload Busy" := "General Preparation"."Tipper 1"."CIP Request", IN_Prod_Ready := "Tipper1 to MB".Product_Ready, IN_Prod_LineOpen := "Tipper1 to MB".Product_LineOpen, IN_SupplyOn := "Tipper1 to MB".Product_SupplyON, IN_Prod_Transfer_Comp := "Tipper1 to MB".Product_Transfer_Complete, "CIP Pulse" := "Timer 5S/30s", "CIP Complete" := "CIP_to_Mix".CIP_Complete."Chili Awetan"."T-02.00_CIP_Complete", Out_AV_Inload =>, Out_AV_Outlet =>, Out_AV_Transfer =>, Out_AV_CIP_Tank =>, Out_AV_CIP_Line =>, Out_P_Inload =>, Out_P_Inload_Sp =>, Out_P_Transfer =>, Out_P_Transfer_Sp =>, Out_P_CIP =>, Out_P_CIP_Sp =>, Out_Prod_Req => "MB to Tipper1".Product_Request, Out_Prod_LineOpen => "MB to Tipper1".Product_Line_OK, Out_CIP_Req => "Mix_to_CIP".CIP_Request."Chili Awetan"."T-02.00_CIP_Request", Out_CIP_LineOpen => "Mix_to_CIP".CIP_Line_OK."Chili Awetan"."T-02.00_CIP_LineOK")
   END_RUNG
   RUNG wire#powerrail
      Contact( "CIP_to_Mix".CIP_Supply_On."Chili Awetan"."T-02.00_CIP_Supply_ON" )
      I_Contact( "General Preparation".CIP_Bypass )
   END_RUNG wire#w1
   RUNG wire#powerrail
      Contact( "General Preparation".CIP_Bypass )
   END_RUNG wire#w1
   RUNG wire#powerrail
      Contact( "CIP_to_Mix".CIP_RequestOK."Chili Awetan"."T-02.00_CIP_RequestOK" )
      I_Contact( "General Preparation".CIP_Bypass )
   END_RUNG wire#w2
   RUNG wire#powerrail
      Contact( "General Preparation".CIP_Bypass )
   END_RUNG wire#w2
   RUNG wire#powerrail
      Contact( "T-03_ChiliAwetan_2".Out_CIP_Req )
   END_RUNG wire#w3
   RUNG wire#powerrail
      Contact( "T-04_ChiliAwetan_3".Out_CIP_Req )
   END_RUNG wire#w3
   RUNG wire#powerrail
      Contact( "T-09_Garlic".Out_CIP_Req )
   END_RUNG wire#w3
   RUNG wire#powerrail
      Contact( "T-10_Vinegar".Out_CIP_Req )
   END_RUNG wire#w3
   RUNG wire#powerrail
      Contact( "General Preparation"."Tipper 1"."CIP Request" )
      Contact( "Mix_to_CIP".CIP_Request.Osa_CIP_Req )
   END_RUNG wire#w3
   RUNG wire#powerrail
      Contact( "General Preparation"."Header 1"."CIP Request" )
   END_RUNG wire#w3
   RUNG wire#powerrail
      Contact( "General Preparation"."Header 2"."CIP Request" )
   END_RUNG wire#w3
   RUNG wire#powerrail
      Contact( "Osa to CIP"."CIP OSA on Process" )
   END_RUNG wire#w3
   // the same network as SCL:
   "T-02_ChiliAwetan_1"(IN_LT01 := "IO Analog Preparation_DB"."LT-02.01".QOUT,   // "BFT_ChiliAwetan"
                        "Inload Busy" := "General Preparation"."Tipper 1"."CIP Request",
                        IN_Prod_Ready := "Tipper1 to MB".Product_Ready,
                        IN_Prod_LineOpen := "Tipper1 to MB".Product_LineOpen,
                        IN_SupplyOn := "Tipper1 to MB".Product_SupplyON,
                        IN_Prod_Transfer_Comp := "Tipper1 to MB".Product_Transfer_Complete,
                        "CIP Pulse" := "Timer 5S/30s",
                        "CIP Supply ON" := ("CIP_to_Mix".CIP_Supply_On."Chili Awetan"."T-02.00_CIP_Supply_ON" AND NOT "General Preparation".CIP_Bypass) OR "General Preparation".CIP_Bypass,
                        "CIP Req OK" := ("CIP_to_Mix".CIP_RequestOK."Chili Awetan"."T-02.00_CIP_RequestOK" AND NOT "General Preparation".CIP_Bypass) OR "General Preparation".CIP_Bypass,
                        "CIP Complete" := "CIP_to_Mix".CIP_Complete."Chili Awetan"."T-02.00_CIP_Complete",
                        "CIP Busy" := "T-03_ChiliAwetan_2".Out_CIP_Req OR "T-04_ChiliAwetan_3".Out_CIP_Req OR "T-09_Garlic".Out_CIP_Req OR "T-10_Vinegar".Out_CIP_Req OR ("General Preparation"."Tipper 1"."CIP Request" AND "Mix_to_CIP".CIP_Request.Osa_CIP_Req) OR "General Preparation"."Header 1"."CIP Request" OR "General Preparation"."Header 2"."CIP Request" OR "Osa to CIP"."CIP OSA on Process",
                        Out_Prod_Req => "MB to Tipper1".Product_Request,
                        Out_Prod_LineOpen => "MB to Tipper1".Product_Line_OK,
                        Out_CIP_Req => "Mix_to_CIP".CIP_Request."Chili Awetan"."T-02.00_CIP_Request",
                        Out_CIP_LineOpen => "Mix_to_CIP".CIP_Line_OK."Chili Awetan"."T-02.00_CIP_LineOK");
END_REGION

REGION Network 13: T-02.00 Valve Cmd
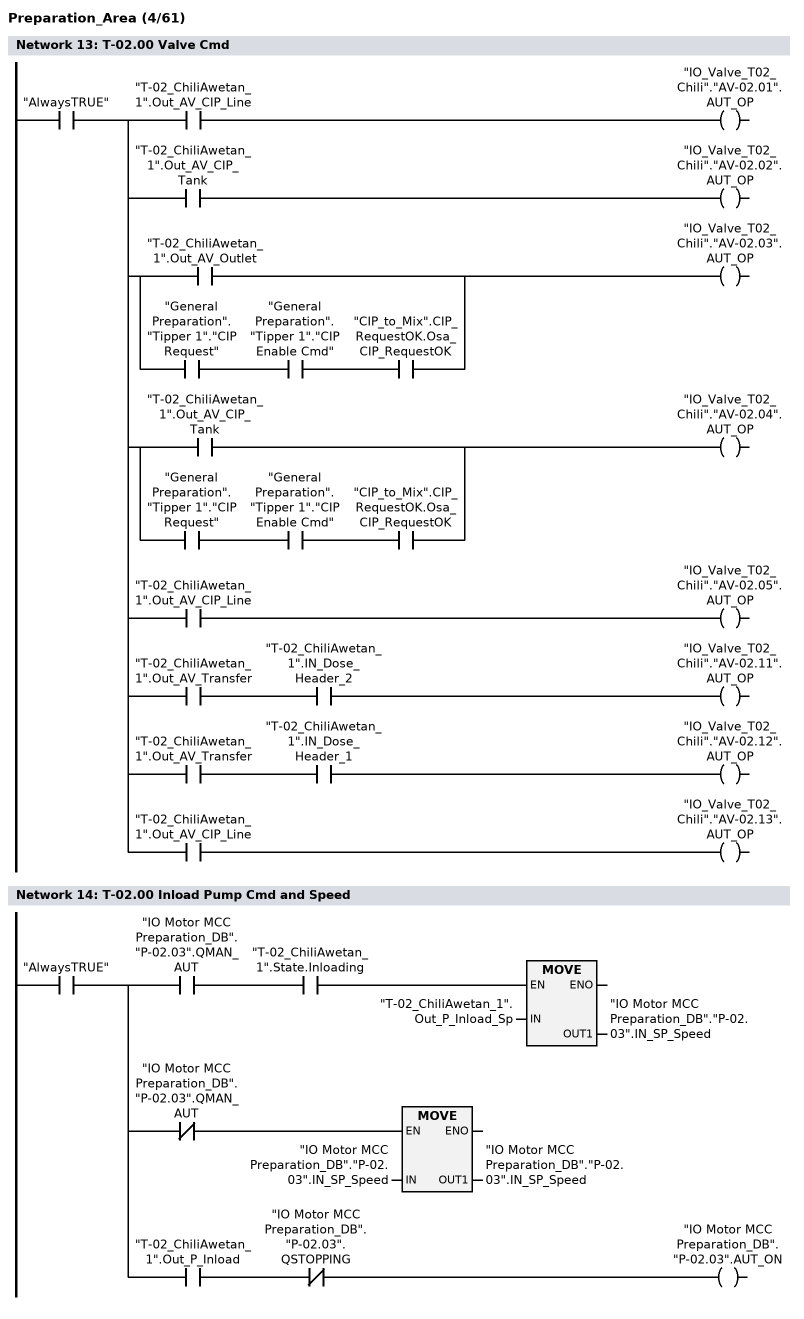
   RUNG wire#powerrail
      Contact( "AlwaysTRUE" )
      wire#w1
      Contact( "T-02_ChiliAwetan_1".Out_AV_CIP_Line )
      Coil( "IO_Valve_T02_Chili"."AV-02.01".AUT_OP )
   END_RUNG
   RUNG wire#w1
      Contact( "T-02_ChiliAwetan_1".Out_AV_CIP_Tank )
      Coil( "IO_Valve_T02_Chili"."AV-02.02".AUT_OP )
   END_RUNG
   RUNG wire#w1
      Contact( "T-02_ChiliAwetan_1".Out_AV_Outlet )
      wire#w2
      Coil( "IO_Valve_T02_Chili"."AV-02.03".AUT_OP )
   END_RUNG
   RUNG wire#w1
      Contact( "General Preparation"."Tipper 1"."CIP Request" )
      Contact( "General Preparation"."Tipper 1"."CIP Enable Cmd" )
      Contact( "CIP_to_Mix".CIP_RequestOK.Osa_CIP_RequestOK )
   END_RUNG wire#w2
   RUNG wire#w1
      Contact( "T-02_ChiliAwetan_1".Out_AV_CIP_Tank )
      wire#w3
      Coil( "IO_Valve_T02_Chili"."AV-02.04".AUT_OP )
   END_RUNG
   RUNG wire#w1
      Contact( "General Preparation"."Tipper 1"."CIP Request" )
      Contact( "General Preparation"."Tipper 1"."CIP Enable Cmd" )
      Contact( "CIP_to_Mix".CIP_RequestOK.Osa_CIP_RequestOK )
   END_RUNG wire#w3
   RUNG wire#w1
      Contact( "T-02_ChiliAwetan_1".Out_AV_CIP_Line )
      Coil( "IO_Valve_T02_Chili"."AV-02.05".AUT_OP )
   END_RUNG
   RUNG wire#w1
      Contact( "T-02_ChiliAwetan_1".Out_AV_Transfer )
      Contact( "T-02_ChiliAwetan_1".IN_Dose_Header_2 )
      Coil( "IO_Valve_T02_Chili"."AV-02.11".AUT_OP )
   END_RUNG
   RUNG wire#w1
      Contact( "T-02_ChiliAwetan_1".Out_AV_Transfer )
      Contact( "T-02_ChiliAwetan_1".IN_Dose_Header_1 )
      Coil( "IO_Valve_T02_Chili"."AV-02.12".AUT_OP )
   END_RUNG
   RUNG wire#w1
      Contact( "T-02_ChiliAwetan_1".Out_AV_CIP_Line )
      Coil( "IO_Valve_T02_Chili"."AV-02.13".AUT_OP )
   END_RUNG
   // the same network as SCL:
   "IO_Valve_T02_Chili"."AV-02.01".AUT_OP := "AlwaysTRUE" AND "T-02_ChiliAwetan_1".Out_AV_CIP_Line;
   "IO_Valve_T02_Chili"."AV-02.02".AUT_OP := "AlwaysTRUE" AND "T-02_ChiliAwetan_1".Out_AV_CIP_Tank;
   "IO_Valve_T02_Chili"."AV-02.03".AUT_OP := "AlwaysTRUE" AND ("T-02_ChiliAwetan_1".Out_AV_Outlet OR ("General Preparation"."Tipper 1"."CIP Request" AND "General Preparation"."Tipper 1"."CIP Enable Cmd" AND "CIP_to_Mix".CIP_RequestOK.Osa_CIP_RequestOK));
   "IO_Valve_T02_Chili"."AV-02.04".AUT_OP := "AlwaysTRUE" AND ("T-02_ChiliAwetan_1".Out_AV_CIP_Tank OR ("General Preparation"."Tipper 1"."CIP Request" AND "General Preparation"."Tipper 1"."CIP Enable Cmd" AND "CIP_to_Mix".CIP_RequestOK.Osa_CIP_RequestOK));
   "IO_Valve_T02_Chili"."AV-02.05".AUT_OP := "AlwaysTRUE" AND "T-02_ChiliAwetan_1".Out_AV_CIP_Line;
   "IO_Valve_T02_Chili"."AV-02.11".AUT_OP := "AlwaysTRUE" AND "T-02_ChiliAwetan_1".Out_AV_Transfer AND "T-02_ChiliAwetan_1".IN_Dose_Header_2;
   "IO_Valve_T02_Chili"."AV-02.12".AUT_OP := "AlwaysTRUE" AND "T-02_ChiliAwetan_1".Out_AV_Transfer AND "T-02_ChiliAwetan_1".IN_Dose_Header_1;
   "IO_Valve_T02_Chili"."AV-02.13".AUT_OP := "AlwaysTRUE" AND "T-02_ChiliAwetan_1".Out_AV_CIP_Line;
END_REGION

REGION Network 14: T-02.00 Inload Pump Cmd and Speed
   RUNG wire#powerrail
      Contact( "AlwaysTRUE" )
      wire#w1
      Contact( "IO Motor MCC Preparation_DB"."P-02.03".QMAN_AUT )
      Contact( "T-02_ChiliAwetan_1".State.Inloading )
      Move(in := "T-02_ChiliAwetan_1".Out_P_Inload_Sp, out1 => "IO Motor MCC Preparation_DB"."P-02.03".IN_SP_Speed)
   END_RUNG
   RUNG wire#w1
      I_Contact( "IO Motor MCC Preparation_DB"."P-02.03".QMAN_AUT )
      Move(in := "IO Motor MCC Preparation_DB"."P-02.03".IN_SP_Speed, out1 => "IO Motor MCC Preparation_DB"."P-02.03".IN_SP_Speed)
   END_RUNG
   RUNG wire#w1
      Contact( "T-02_ChiliAwetan_1".Out_P_Inload )
      I_Contact( "IO Motor MCC Preparation_DB"."P-02.03".QSTOPPING )
      Coil( "IO Motor MCC Preparation_DB"."P-02.03".AUT_ON )
   END_RUNG
   // the same network as SCL:
   IF "AlwaysTRUE" AND "IO Motor MCC Preparation_DB"."P-02.03".QMAN_AUT AND "T-02_ChiliAwetan_1".State.Inloading THEN
       "IO Motor MCC Preparation_DB"."P-02.03".IN_SP_Speed := "T-02_ChiliAwetan_1".Out_P_Inload_Sp;
   END_IF;
   IF "AlwaysTRUE" AND NOT "IO Motor MCC Preparation_DB"."P-02.03".QMAN_AUT THEN
       "IO Motor MCC Preparation_DB"."P-02.03".IN_SP_Speed := "IO Motor MCC Preparation_DB"."P-02.03".IN_SP_Speed;
   END_IF;
   "IO Motor MCC Preparation_DB"."P-02.03".AUT_ON := "AlwaysTRUE" AND "T-02_ChiliAwetan_1".Out_P_Inload AND NOT "IO Motor MCC Preparation_DB"."P-02.03".QSTOPPING;
END_REGION

REGION Network 15: T-02.00 Transfer Pump Cmd and Speed
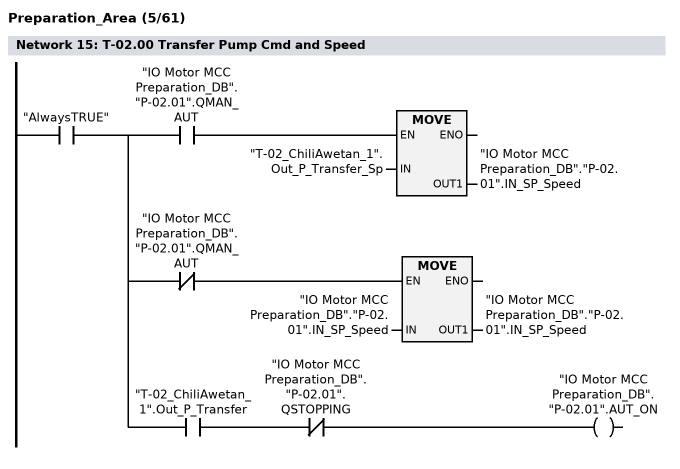
   RUNG wire#powerrail
      Contact( "AlwaysTRUE" )
      wire#w1
      Contact( "IO Motor MCC Preparation_DB"."P-02.01".QMAN_AUT )
      Move(in := "T-02_ChiliAwetan_1".Out_P_Transfer_Sp, out1 => "IO Motor MCC Preparation_DB"."P-02.01".IN_SP_Speed)
   END_RUNG
   RUNG wire#w1
      I_Contact( "IO Motor MCC Preparation_DB"."P-02.01".QMAN_AUT )
      Move(in := "IO Motor MCC Preparation_DB"."P-02.01".IN_SP_Speed, out1 => "IO Motor MCC Preparation_DB"."P-02.01".IN_SP_Speed)
   END_RUNG
   RUNG wire#w1
      Contact( "T-02_ChiliAwetan_1".Out_P_Transfer )
      I_Contact( "IO Motor MCC Preparation_DB"."P-02.01".QSTOPPING )
      Coil( "IO Motor MCC Preparation_DB"."P-02.01".AUT_ON )
   END_RUNG
   // the same network as SCL:
   IF "AlwaysTRUE" AND "IO Motor MCC Preparation_DB"."P-02.01".QMAN_AUT THEN
       "IO Motor MCC Preparation_DB"."P-02.01".IN_SP_Speed := "T-02_ChiliAwetan_1".Out_P_Transfer_Sp;
   END_IF;
   IF "AlwaysTRUE" AND NOT "IO Motor MCC Preparation_DB"."P-02.01".QMAN_AUT THEN
       "IO Motor MCC Preparation_DB"."P-02.01".IN_SP_Speed := "IO Motor MCC Preparation_DB"."P-02.01".IN_SP_Speed;
   END_IF;
   "IO Motor MCC Preparation_DB"."P-02.01".AUT_ON := "AlwaysTRUE" AND "T-02_ChiliAwetan_1".Out_P_Transfer AND NOT "IO Motor MCC Preparation_DB"."P-02.01".QSTOPPING;
END_REGION

REGION Network 16: T-02.00 Feedback Instrument
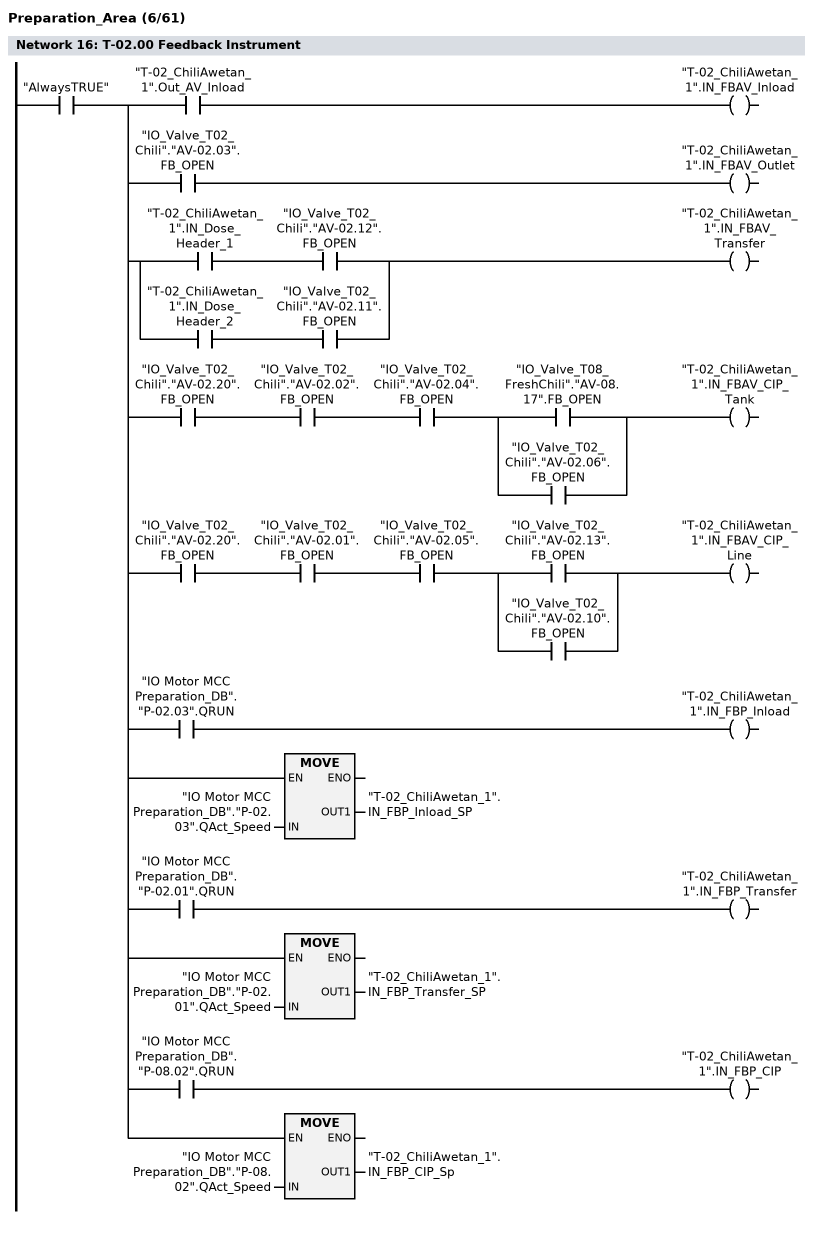
   RUNG wire#powerrail
      Contact( "AlwaysTRUE" )
      wire#w1
      Contact( "T-02_ChiliAwetan_1".Out_AV_Inload )
      Coil( "T-02_ChiliAwetan_1".IN_FBAV_Inload )
   END_RUNG
   RUNG wire#w1
      Contact( "IO_Valve_T02_Chili"."AV-02.03".FB_OPEN )
      Coil( "T-02_ChiliAwetan_1".IN_FBAV_Outlet )
   END_RUNG
   RUNG wire#w1
      Contact( "T-02_ChiliAwetan_1".IN_Dose_Header_1 )
      Contact( "IO_Valve_T02_Chili"."AV-02.12".FB_OPEN )
      wire#w2
      Coil( "T-02_ChiliAwetan_1".IN_FBAV_Transfer )
   END_RUNG
   RUNG wire#w1
      Contact( "T-02_ChiliAwetan_1".IN_Dose_Header_2 )
      Contact( "IO_Valve_T02_Chili"."AV-02.11".FB_OPEN )
   END_RUNG wire#w2
   RUNG wire#w1
      Contact( "IO_Valve_T02_Chili"."AV-02.20".FB_OPEN )
      Contact( "IO_Valve_T02_Chili"."AV-02.02".FB_OPEN )
      Contact( "IO_Valve_T02_Chili"."AV-02.04".FB_OPEN )
      wire#w3
      Contact( "IO_Valve_T08_FreshChili"."AV-08.17".FB_OPEN )
      wire#w4
      Coil( "T-02_ChiliAwetan_1".IN_FBAV_CIP_Tank )
   END_RUNG
   RUNG wire#w3
      Contact( "IO_Valve_T02_Chili"."AV-02.06".FB_OPEN )
   END_RUNG wire#w4
   RUNG wire#w1
      Contact( "IO_Valve_T02_Chili"."AV-02.20".FB_OPEN )
      Contact( "IO_Valve_T02_Chili"."AV-02.01".FB_OPEN )
      Contact( "IO_Valve_T02_Chili"."AV-02.05".FB_OPEN )
      wire#w5
      Contact( "IO_Valve_T02_Chili"."AV-02.13".FB_OPEN )
      wire#w6
      Coil( "T-02_ChiliAwetan_1".IN_FBAV_CIP_Line )
   END_RUNG
   RUNG wire#w5
      Contact( "IO_Valve_T02_Chili"."AV-02.10".FB_OPEN )
   END_RUNG wire#w6
   RUNG wire#w1
      Contact( "IO Motor MCC Preparation_DB"."P-02.03".QRUN )
      Coil( "T-02_ChiliAwetan_1".IN_FBP_Inload )
   END_RUNG
   RUNG wire#w1
      Move(in := "IO Motor MCC Preparation_DB"."P-02.03".QAct_Speed, out1 => "T-02_ChiliAwetan_1".IN_FBP_Inload_SP)
   END_RUNG
   RUNG wire#w1
      Contact( "IO Motor MCC Preparation_DB"."P-02.01".QRUN )
      Coil( "T-02_ChiliAwetan_1".IN_FBP_Transfer )
   END_RUNG
   RUNG wire#w1
      Move(in := "IO Motor MCC Preparation_DB"."P-02.01".QAct_Speed, out1 => "T-02_ChiliAwetan_1".IN_FBP_Transfer_SP)
   END_RUNG
   RUNG wire#w1
      Contact( "IO Motor MCC Preparation_DB"."P-08.02".QRUN )
      Coil( "T-02_ChiliAwetan_1".IN_FBP_CIP )
   END_RUNG
   RUNG wire#w1
      Move(in := "IO Motor MCC Preparation_DB"."P-08.02".QAct_Speed, out1 => "T-02_ChiliAwetan_1".IN_FBP_CIP_Sp)
   END_RUNG
   // the same network as SCL:
   "T-02_ChiliAwetan_1".IN_FBAV_Inload := "AlwaysTRUE" AND "T-02_ChiliAwetan_1".Out_AV_Inload;
   "T-02_ChiliAwetan_1".IN_FBAV_Outlet := "AlwaysTRUE" AND "IO_Valve_T02_Chili"."AV-02.03".FB_OPEN;
   "T-02_ChiliAwetan_1".IN_FBAV_Transfer := "AlwaysTRUE" AND (("T-02_ChiliAwetan_1".IN_Dose_Header_1 AND "IO_Valve_T02_Chili"."AV-02.12".FB_OPEN) OR ("T-02_ChiliAwetan_1".IN_Dose_Header_2 AND "IO_Valve_T02_Chili"."AV-02.11".FB_OPEN));
   "T-02_ChiliAwetan_1".IN_FBAV_CIP_Tank := "AlwaysTRUE" AND "IO_Valve_T02_Chili"."AV-02.20".FB_OPEN AND "IO_Valve_T02_Chili"."AV-02.02".FB_OPEN AND "IO_Valve_T02_Chili"."AV-02.04".FB_OPEN AND ("IO_Valve_T08_FreshChili"."AV-08.17".FB_OPEN OR "IO_Valve_T02_Chili"."AV-02.06".FB_OPEN);
   "T-02_ChiliAwetan_1".IN_FBAV_CIP_Line := "AlwaysTRUE" AND "IO_Valve_T02_Chili"."AV-02.20".FB_OPEN AND "IO_Valve_T02_Chili"."AV-02.01".FB_OPEN AND "IO_Valve_T02_Chili"."AV-02.05".FB_OPEN AND ("IO_Valve_T02_Chili"."AV-02.13".FB_OPEN OR "IO_Valve_T02_Chili"."AV-02.10".FB_OPEN);
   "T-02_ChiliAwetan_1".IN_FBP_Inload := "AlwaysTRUE" AND "IO Motor MCC Preparation_DB"."P-02.03".QRUN;
   IF "AlwaysTRUE" THEN
       "T-02_ChiliAwetan_1".IN_FBP_Inload_SP := "IO Motor MCC Preparation_DB"."P-02.03".QAct_Speed;
   END_IF;
   "T-02_ChiliAwetan_1".IN_FBP_Transfer := "AlwaysTRUE" AND "IO Motor MCC Preparation_DB"."P-02.01".QRUN;
   IF "AlwaysTRUE" THEN
       "T-02_ChiliAwetan_1".IN_FBP_Transfer_SP := "IO Motor MCC Preparation_DB"."P-02.01".QAct_Speed;
   END_IF;
   "T-02_ChiliAwetan_1".IN_FBP_CIP := "AlwaysTRUE" AND "IO Motor MCC Preparation_DB"."P-08.02".QRUN;
   IF "AlwaysTRUE" THEN
       "T-02_ChiliAwetan_1".IN_FBP_CIP_Sp := "IO Motor MCC Preparation_DB"."P-08.02".QAct_Speed;
   END_IF;
END_REGION

REGION Network 17: T-02.00 Comm to Blend
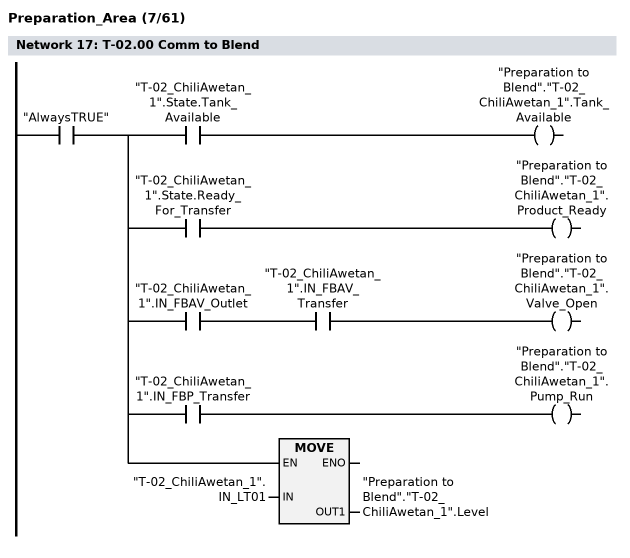
   RUNG wire#powerrail
      Contact( "AlwaysTRUE" )
      wire#w1
      Contact( "T-02_ChiliAwetan_1".State.Tank_Available )
      Coil( "Preparation to Blend"."T-02_ChiliAwetan_1".Tank_Available )
   END_RUNG
   RUNG wire#w1
      Contact( "T-02_ChiliAwetan_1".State.Ready_For_Transfer )
      Coil( "Preparation to Blend"."T-02_ChiliAwetan_1".Product_Ready )
   END_RUNG
   RUNG wire#w1
      Contact( "T-02_ChiliAwetan_1".IN_FBAV_Outlet )
      Contact( "T-02_ChiliAwetan_1".IN_FBAV_Transfer )
      Coil( "Preparation to Blend"."T-02_ChiliAwetan_1".Valve_Open )
   END_RUNG
   RUNG wire#w1
      Contact( "T-02_ChiliAwetan_1".IN_FBP_Transfer )
      Coil( "Preparation to Blend"."T-02_ChiliAwetan_1".Pump_Run )
   END_RUNG
   RUNG wire#w1
      Move(in := "T-02_ChiliAwetan_1".IN_LT01, out1 => "Preparation to Blend"."T-02_ChiliAwetan_1".Level)
   END_RUNG
   // the same network as SCL:
   "Preparation to Blend"."T-02_ChiliAwetan_1".Tank_Available := "AlwaysTRUE" AND "T-02_ChiliAwetan_1".State.Tank_Available;
   "Preparation to Blend"."T-02_ChiliAwetan_1".Product_Ready := "AlwaysTRUE" AND "T-02_ChiliAwetan_1".State.Ready_For_Transfer;
   "Preparation to Blend"."T-02_ChiliAwetan_1".Valve_Open := "AlwaysTRUE" AND "T-02_ChiliAwetan_1".IN_FBAV_Outlet AND "T-02_ChiliAwetan_1".IN_FBAV_Transfer;
   "Preparation to Blend"."T-02_ChiliAwetan_1".Pump_Run := "AlwaysTRUE" AND "T-02_ChiliAwetan_1".IN_FBP_Transfer;
   IF "AlwaysTRUE" THEN
       "Preparation to Blend"."T-02_ChiliAwetan_1".Level := "T-02_ChiliAwetan_1".IN_LT01;
   END_IF;
END_REGION

NETWORK
TITLE = T-03.00 DOSE ON OFF
      O     "Blend to Preparation"."T-20".Raw_Material.ChiliAwetan_2.DoseRun;
      O     "Blend to Preparation"."T-21".Raw_Material.ChiliAwetan_2.DoseRun;
      O     "Blend to Preparation"."T-30".Raw_Material.ChiliAwetan_2.DoseRun;
      O     "Blend to Preparation"."T-31".Raw_Material.ChiliAwetan_2.DoseRun;
      O     "Blend to Preparation"."T-40".Raw_Material.ChiliAwetan_2.DoseRun;
      O     "Blend to Preparation"."T-41".Raw_Material.ChiliAwetan_2.DoseRun;
      =     "T-03_ChiliAwetan_2".IN_Dose_Run;

NETWORK
TITLE = T-03.00 DOSE PAUSE
      O     "Blend to Preparation"."T-20".Raw_Material.ChiliAwetan_2.DoseHeld;
      O     "Blend to Preparation"."T-21".Raw_Material.ChiliAwetan_2.DoseHeld;
      O     "Blend to Preparation"."T-30".Raw_Material.ChiliAwetan_2.DoseHeld;
      O     "Blend to Preparation"."T-31".Raw_Material.ChiliAwetan_2.DoseHeld;
      O     "Blend to Preparation"."T-40".Raw_Material.ChiliAwetan_2.DoseHeld;
      O     "Blend to Preparation"."T-41".Raw_Material.ChiliAwetan_2.DoseHeld;
      =     "T-03_ChiliAwetan_2".IN_Dose_Held;

NETWORK
TITLE = T-03.00 DOSE VALVE CMD
      O(;
      A     "Blend to Preparation"."T-20".Raw_Material.ChiliAwetan_2.DoseRun;
      A     "Blend to Preparation"."T-20".Raw_Material.ChiliAwetan_2.ValveCMD;
      );
      O(;
      A     "Blend to Preparation"."T-21".Raw_Material.ChiliAwetan_2.DoseRun;
      A     "Blend to Preparation"."T-21".Raw_Material.ChiliAwetan_2.ValveCMD;
      );
      O(;
      A     "Blend to Preparation"."T-30".Raw_Material.ChiliAwetan_2.DoseRun;
      A     "Blend to Preparation"."T-30".Raw_Material.ChiliAwetan_2.ValveCMD;
      );
      O(;
      A     "Blend to Preparation"."T-31".Raw_Material.ChiliAwetan_2.DoseRun;
      A     "Blend to Preparation"."T-31".Raw_Material.ChiliAwetan_2.ValveCMD;
      );
      O(;
      A     "Blend to Preparation"."T-40".Raw_Material.ChiliAwetan_2.DoseRun;
      A     "Blend to Preparation"."T-40".Raw_Material.ChiliAwetan_2.ValveCMD;
      );
      O(;
      A     "Blend to Preparation"."T-41".Raw_Material.ChiliAwetan_2.DoseRun;
      A     "Blend to Preparation"."T-41".Raw_Material.ChiliAwetan_2.ValveCMD;
      );
      =     "T-03_ChiliAwetan_2".IN_Dose_Valve_Cmd;


NETWORK
TITLE = T-03.00 DOSE Pump CMD
      O(;
      A     "Blend to Preparation"."T-20".Raw_Material.ChiliAwetan_2.DoseRun;
      A     "Blend to Preparation"."T-20".Raw_Material.ChiliAwetan_2.PumpCMD;
      );
      O(;
      A     "Blend to Preparation"."T-21".Raw_Material.ChiliAwetan_2.DoseRun;
      A     "Blend to Preparation"."T-21".Raw_Material.ChiliAwetan_2.PumpCMD;
      );
      O(;
      A     "Blend to Preparation"."T-30".Raw_Material.ChiliAwetan_2.DoseRun;
      A     "Blend to Preparation"."T-30".Raw_Material.ChiliAwetan_2.PumpCMD;
      );
      O(;
      A     "Blend to Preparation"."T-31".Raw_Material.ChiliAwetan_2.DoseRun;
      A     "Blend to Preparation"."T-31".Raw_Material.ChiliAwetan_2.PumpCMD;
      );
      O(;
      A     "Blend to Preparation"."T-40".Raw_Material.ChiliAwetan_2.DoseRun;
      A     "Blend to Preparation"."T-40".Raw_Material.ChiliAwetan_2.PumpCMD;
      );
      O(;
      A     "Blend to Preparation"."T-41".Raw_Material.ChiliAwetan_2.DoseRun;
      A     "Blend to Preparation"."T-41".Raw_Material.ChiliAwetan_2.PumpCMD;
      );
      =     "T-03_ChiliAwetan_2".IN_Dose_Pump_Cmd;



NETWORK
TITLE = T-03.00 DOSE PUMP SPEED
// Checking
      O     "Blend to Preparation"."T-20".Raw_Material.ChiliAwetan_2.DoseRun;
      JC    SP_03_FROM_20;
      O     "Blend to Preparation"."T-21".Raw_Material.ChiliAwetan_2.DoseRun;
      JC    SP_03_FROM_21;
      O     "Blend to Preparation"."T-30".Raw_Material.ChiliAwetan_2.DoseRun;
      JC    SP_03_FROM_30;
      O     "Blend to Preparation"."T-31".Raw_Material.ChiliAwetan_2.DoseRun;
      JC    SP_03_FROM_31;
      O     "Blend to Preparation"."T-40".Raw_Material.ChiliAwetan_2.DoseRun;
      JC    SP_03_FROM_40;
      O     "Blend to Preparation"."T-41".Raw_Material.ChiliAwetan_2.DoseRun;
      JC    SP_03_FROM_41;
//Jump to end if Blend not Dosing
      JC    SP_03_SELF;
//Load Set Point
SP_03_FROM_20:L     "Blend to Preparation".Recipe."T-20".ChiliAwetan_2.SP_PumpSpeed;
      T     "T-03_ChiliAwetan_2".IN_Dose_Pump_Sp;
      JC    SP_03_SELF;
SP_03_FROM_21:L     "Blend to Preparation".Recipe."T-21".ChiliAwetan_2.SP_PumpSpeed;
      T     "T-03_ChiliAwetan_2".IN_Dose_Pump_Sp;
      JC    SP_03_SELF;
SP_03_FROM_30:L     "Blend to Preparation".Recipe."T-30".ChiliAwetan_2.SP_PumpSpeed;
      T     "T-03_ChiliAwetan_2".IN_Dose_Pump_Sp;
      JC    SP_03_SELF;
SP_03_FROM_31:L     "Blend to Preparation".Recipe."T-31".ChiliAwetan_2.SP_PumpSpeed;
      T     "T-03_ChiliAwetan_2".IN_Dose_Pump_Sp;
      JC    SP_03_SELF;
SP_03_FROM_40:L     "Blend to Preparation".Recipe."T-40".ChiliAwetan_2.SP_PumpSpeed;
      T     "T-03_ChiliAwetan_2".IN_Dose_Pump_Sp;
      JC    SP_03_SELF;
SP_03_FROM_41:L     "Blend to Preparation".Recipe."T-41".ChiliAwetan_2.SP_PumpSpeed;
      T     "T-03_ChiliAwetan_2".IN_Dose_Pump_Sp;
      JC    SP_03_SELF;
// END
SP_03_SELF:L     "T-03_ChiliAwetan_2".IN_Dose_Pump_Sp;
      T     "T-03_ChiliAwetan_2".IN_Dose_Pump_Sp;


NETWORK
TITLE = T-03.00 Header Req
// HEADER 1 Req
      O     "Blend to Preparation"."T-20".Raw_Material.ChiliAwetan_2.Header1_Req;
      O     "Blend to Preparation"."T-21".Raw_Material.ChiliAwetan_2.Header1_Req;
      O     "Blend to Preparation"."T-30".Raw_Material.ChiliAwetan_2.Header1_Req;
      O     "Blend to Preparation"."T-31".Raw_Material.ChiliAwetan_2.Header1_Req;
      O     "Blend to Preparation"."T-40".Raw_Material.ChiliAwetan_2.Header1_Req;
      O     "Blend to Preparation"."T-41".Raw_Material.ChiliAwetan_2.Header1_Req;
      =     "T-03_ChiliAwetan_2".IN_Dose_Header_1;

// HEADER 2 Req
      O     "Blend to Preparation"."T-20".Raw_Material.ChiliAwetan_2.Header2_Req;
      O     "Blend to Preparation"."T-21".Raw_Material.ChiliAwetan_2.Header2_Req;
      O     "Blend to Preparation"."T-30".Raw_Material.ChiliAwetan_2.Header2_Req;
      O     "Blend to Preparation"."T-31".Raw_Material.ChiliAwetan_2.Header2_Req;
      O     "Blend to Preparation"."T-40".Raw_Material.ChiliAwetan_2.Header2_Req;
      O     "Blend to Preparation"."T-41".Raw_Material.ChiliAwetan_2.Header2_Req;
      =     "T-03_ChiliAwetan_2".IN_Dose_Header_2;


REGION Network 26: T-03.00 LineTransferOK
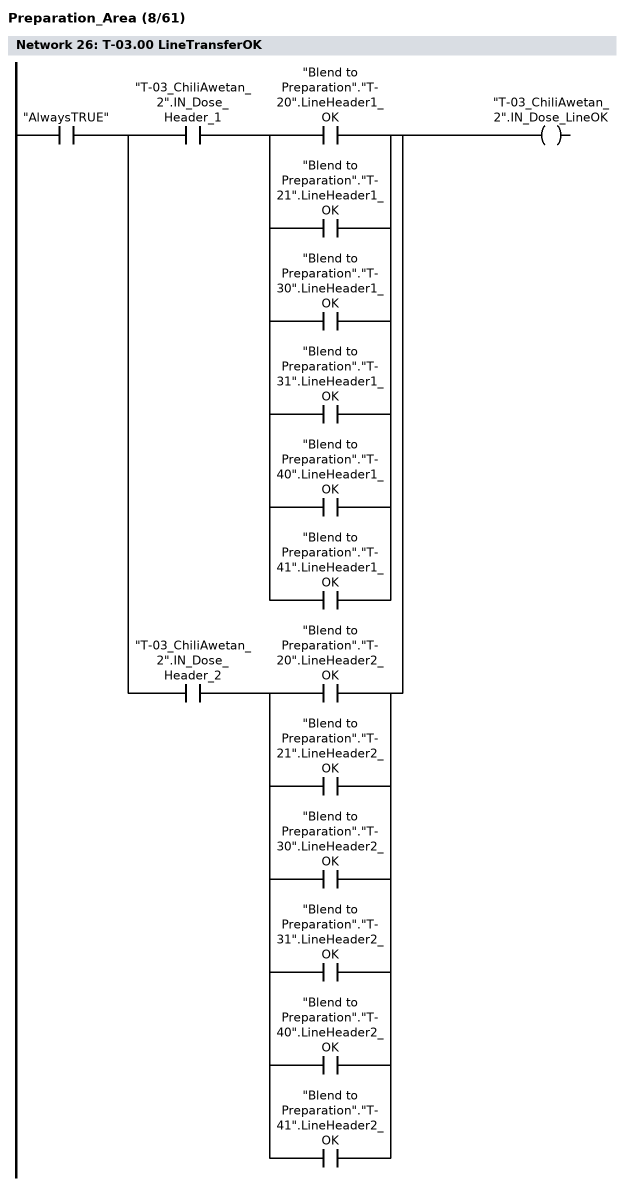
   RUNG wire#powerrail
      Contact( "AlwaysTRUE" )
      wire#w1
      Contact( "T-03_ChiliAwetan_2".IN_Dose_Header_1 )
      wire#w2
      Contact( "Blend to Preparation"."T-20".LineHeader1_OK )
      wire#w3
      Coil( "T-03_ChiliAwetan_2".IN_Dose_LineOK )
   END_RUNG
   RUNG wire#w2
      Contact( "Blend to Preparation"."T-21".LineHeader1_OK )
   END_RUNG wire#w3
   RUNG wire#w2
      Contact( "Blend to Preparation"."T-30".LineHeader1_OK )
   END_RUNG wire#w3
   RUNG wire#w2
      Contact( "Blend to Preparation"."T-31".LineHeader1_OK )
   END_RUNG wire#w3
   RUNG wire#w2
      Contact( "Blend to Preparation"."T-40".LineHeader1_OK )
   END_RUNG wire#w3
   RUNG wire#w2
      Contact( "Blend to Preparation"."T-41".LineHeader1_OK )
   END_RUNG wire#w3
   RUNG wire#w1
      Contact( "T-03_ChiliAwetan_2".IN_Dose_Header_2 )
      wire#w4
      Contact( "Blend to Preparation"."T-20".LineHeader2_OK )
   END_RUNG wire#w3
   RUNG wire#w4
      Contact( "Blend to Preparation"."T-21".LineHeader2_OK )
   END_RUNG wire#w3
   RUNG wire#w4
      Contact( "Blend to Preparation"."T-30".LineHeader2_OK )
   END_RUNG wire#w3
   RUNG wire#w4
      Contact( "Blend to Preparation"."T-31".LineHeader2_OK )
   END_RUNG wire#w3
   RUNG wire#w4
      Contact( "Blend to Preparation"."T-40".LineHeader2_OK )
   END_RUNG wire#w3
   RUNG wire#w4
      Contact( "Blend to Preparation"."T-41".LineHeader2_OK )
   END_RUNG wire#w3
   // the same network as SCL:
   "T-03_ChiliAwetan_2".IN_Dose_LineOK := "AlwaysTRUE" AND (("T-03_ChiliAwetan_2".IN_Dose_Header_1 AND ("Blend to Preparation"."T-20".LineHeader1_OK OR "Blend to Preparation"."T-21".LineHeader1_OK OR "Blend to Preparation"."T-30".LineHeader1_OK OR "Blend to Preparation"."T-31".LineHeader1_OK OR "Blend to Preparation"."T-40".LineHeader1_OK OR "Blend to Preparation"."T-41".LineHeader1_OK)) OR ("T-03_ChiliAwetan_2".IN_Dose_Header_2 AND ("Blend to Preparation"."T-20".LineHeader2_OK OR "Blend to Preparation"."T-21".LineHeader2_OK OR "Blend to Preparation"."T-30".LineHeader2_OK OR "Blend to Preparation"."T-31".LineHeader2_OK OR "Blend to Preparation"."T-40".LineHeader2_OK OR "Blend to Preparation"."T-41".LineHeader2_OK)));
END_REGION

REGION Network 27: T-03.00___Chili Awetan 2
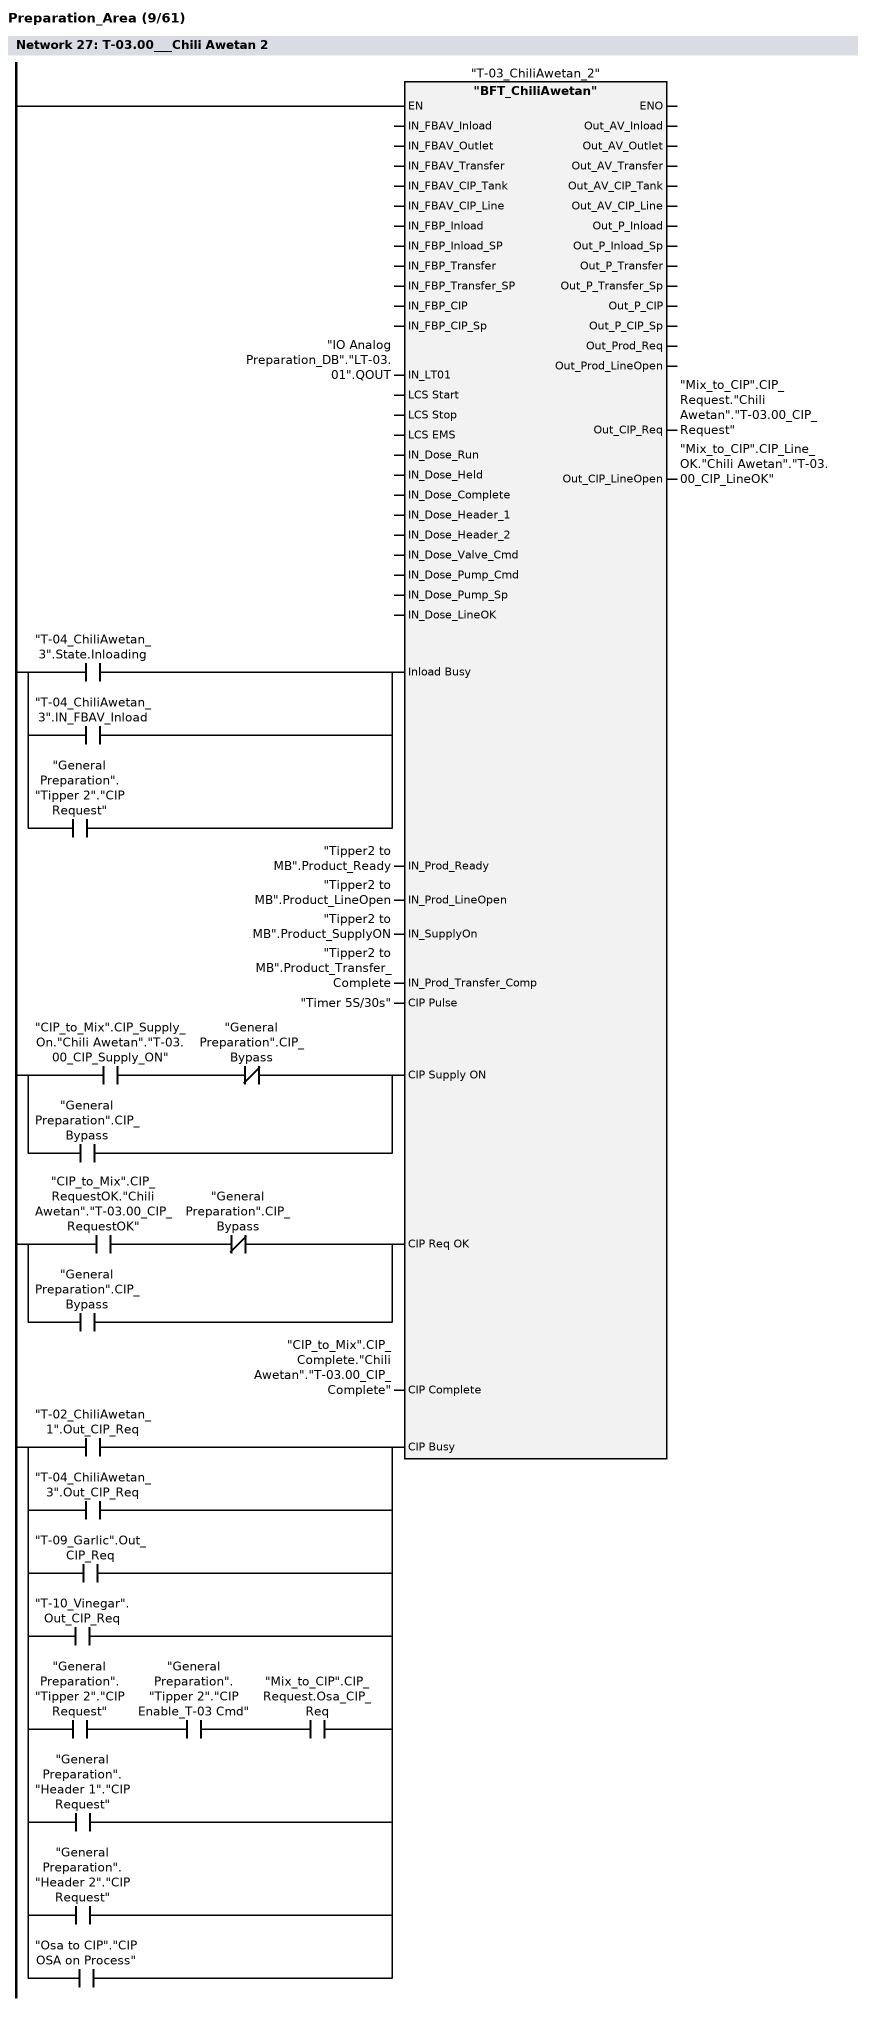
   RUNG wire#powerrail
      "T-03_ChiliAwetan_2"("Inload Busy" := wire#w1, "CIP Supply ON" := wire#w2, "CIP Req OK" := wire#w3, "CIP Busy" := wire#w4, IN_FBAV_Inload :=, IN_FBAV_Outlet :=, IN_FBAV_Transfer :=, IN_FBAV_CIP_Tank :=, IN_FBAV_CIP_Line :=, IN_FBP_Inload :=, IN_FBP_Inload_SP :=, IN_FBP_Transfer :=, IN_FBP_Transfer_SP :=, IN_FBP_CIP :=, IN_FBP_CIP_Sp :=, IN_LT01 := "IO Analog Preparation_DB"."LT-03.01".QOUT, "LCS Start" :=, "LCS Stop" :=, "LCS EMS" :=, IN_Dose_Run :=, IN_Dose_Held :=, IN_Dose_Complete :=, IN_Dose_Header_1 :=, IN_Dose_Header_2 :=, IN_Dose_Valve_Cmd :=, IN_Dose_Pump_Cmd :=, IN_Dose_Pump_Sp :=, IN_Dose_LineOK :=, IN_Prod_Ready := "Tipper2 to MB".Product_Ready, IN_Prod_LineOpen := "Tipper2 to MB".Product_LineOpen, IN_SupplyOn := "Tipper2 to MB".Product_SupplyON, IN_Prod_Transfer_Comp := "Tipper2 to MB".Product_Transfer_Complete, "CIP Pulse" := "Timer 5S/30s", "CIP Complete" := "CIP_to_Mix".CIP_Complete."Chili Awetan"."T-03.00_CIP_Complete", Out_AV_Inload =>, Out_AV_Outlet =>, Out_AV_Transfer =>, Out_AV_CIP_Tank =>, Out_AV_CIP_Line =>, Out_P_Inload =>, Out_P_Inload_Sp =>, Out_P_Transfer =>, Out_P_Transfer_Sp =>, Out_P_CIP =>, Out_P_CIP_Sp =>, Out_Prod_Req =>, Out_Prod_LineOpen =>, Out_CIP_Req => "Mix_to_CIP".CIP_Request."Chili Awetan"."T-03.00_CIP_Request", Out_CIP_LineOpen => "Mix_to_CIP".CIP_Line_OK."Chili Awetan"."T-03.00_CIP_LineOK")
   END_RUNG
   RUNG wire#powerrail
      Contact( "T-04_ChiliAwetan_3".State.Inloading )
   END_RUNG wire#w1
   RUNG wire#powerrail
      Contact( "T-04_ChiliAwetan_3".IN_FBAV_Inload )
   END_RUNG wire#w1
   RUNG wire#powerrail
      Contact( "General Preparation"."Tipper 2"."CIP Request" )
   END_RUNG wire#w1
   RUNG wire#powerrail
      Contact( "CIP_to_Mix".CIP_Supply_On."Chili Awetan"."T-03.00_CIP_Supply_ON" )
      I_Contact( "General Preparation".CIP_Bypass )
   END_RUNG wire#w2
   RUNG wire#powerrail
      Contact( "General Preparation".CIP_Bypass )
   END_RUNG wire#w2
   RUNG wire#powerrail
      Contact( "CIP_to_Mix".CIP_RequestOK."Chili Awetan"."T-03.00_CIP_RequestOK" )
      I_Contact( "General Preparation".CIP_Bypass )
   END_RUNG wire#w3
   RUNG wire#powerrail
      Contact( "General Preparation".CIP_Bypass )
   END_RUNG wire#w3
   RUNG wire#powerrail
      Contact( "T-02_ChiliAwetan_1".Out_CIP_Req )
   END_RUNG wire#w4
   RUNG wire#powerrail
      Contact( "T-04_ChiliAwetan_3".Out_CIP_Req )
   END_RUNG wire#w4
   RUNG wire#powerrail
      Contact( "T-09_Garlic".Out_CIP_Req )
   END_RUNG wire#w4
   RUNG wire#powerrail
      Contact( "T-10_Vinegar".Out_CIP_Req )
   END_RUNG wire#w4
   RUNG wire#powerrail
      Contact( "General Preparation"."Tipper 2"."CIP Request" )
      Contact( "General Preparation"."Tipper 2"."CIP Enable_T-03 Cmd" )
      Contact( "Mix_to_CIP".CIP_Request.Osa_CIP_Req )
   END_RUNG wire#w4
   RUNG wire#powerrail
      Contact( "General Preparation"."Header 1"."CIP Request" )
   END_RUNG wire#w4
   RUNG wire#powerrail
      Contact( "General Preparation"."Header 2"."CIP Request" )
   END_RUNG wire#w4
   RUNG wire#powerrail
      Contact( "Osa to CIP"."CIP OSA on Process" )
   END_RUNG wire#w4
   // the same network as SCL:
   "T-03_ChiliAwetan_2"(IN_LT01 := "IO Analog Preparation_DB"."LT-03.01".QOUT,   // "BFT_ChiliAwetan"
                        "Inload Busy" := "T-04_ChiliAwetan_3".State.Inloading OR "T-04_ChiliAwetan_3".IN_FBAV_Inload OR "General Preparation"."Tipper 2"."CIP Request",
                        IN_Prod_Ready := "Tipper2 to MB".Product_Ready,
                        IN_Prod_LineOpen := "Tipper2 to MB".Product_LineOpen,
                        IN_SupplyOn := "Tipper2 to MB".Product_SupplyON,
                        IN_Prod_Transfer_Comp := "Tipper2 to MB".Product_Transfer_Complete,
                        "CIP Pulse" := "Timer 5S/30s",
                        "CIP Supply ON" := ("CIP_to_Mix".CIP_Supply_On."Chili Awetan"."T-03.00_CIP_Supply_ON" AND NOT "General Preparation".CIP_Bypass) OR "General Preparation".CIP_Bypass,
                        "CIP Req OK" := ("CIP_to_Mix".CIP_RequestOK."Chili Awetan"."T-03.00_CIP_RequestOK" AND NOT "General Preparation".CIP_Bypass) OR "General Preparation".CIP_Bypass,
                        "CIP Complete" := "CIP_to_Mix".CIP_Complete."Chili Awetan"."T-03.00_CIP_Complete",
                        "CIP Busy" := "T-02_ChiliAwetan_1".Out_CIP_Req OR "T-04_ChiliAwetan_3".Out_CIP_Req OR "T-09_Garlic".Out_CIP_Req OR "T-10_Vinegar".Out_CIP_Req OR ("General Preparation"."Tipper 2"."CIP Request" AND "General Preparation"."Tipper 2"."CIP Enable_T-03 Cmd" AND "Mix_to_CIP".CIP_Request.Osa_CIP_Req) OR "General Preparation"."Header 1"."CIP Request" OR "General Preparation"."Header 2"."CIP Request" OR "Osa to CIP"."CIP OSA on Process",
                        Out_CIP_Req => "Mix_to_CIP".CIP_Request."Chili Awetan"."T-03.00_CIP_Request",
                        Out_CIP_LineOpen => "Mix_to_CIP".CIP_Line_OK."Chili Awetan"."T-03.00_CIP_LineOK");
END_REGION

REGION Network 28: T-03.00 Valve Cmd
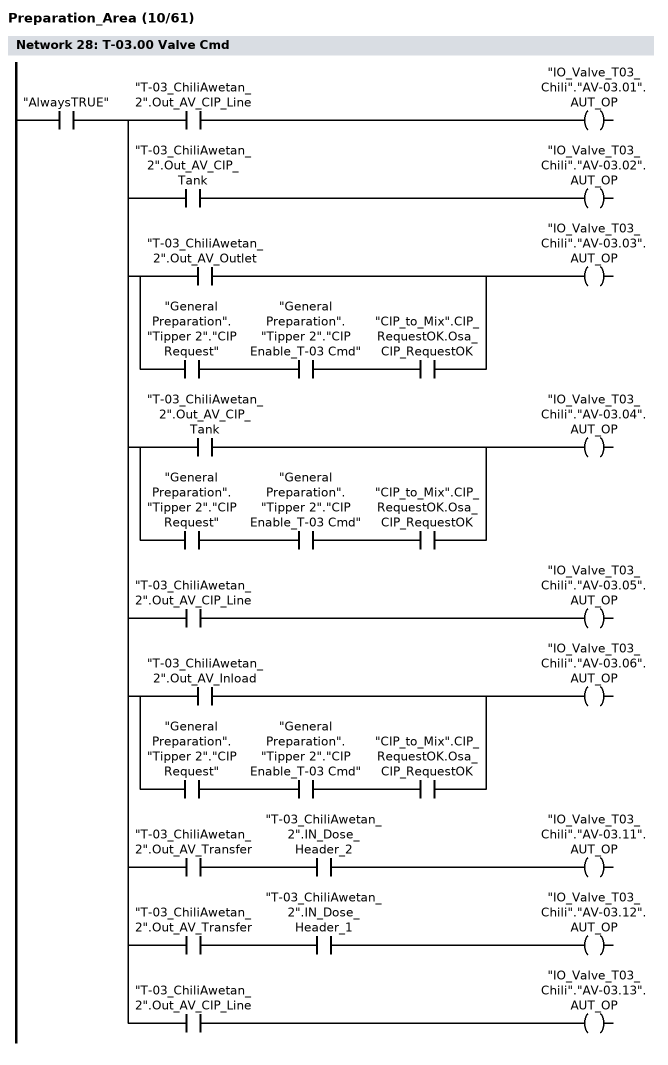
   RUNG wire#powerrail
      Contact( "AlwaysTRUE" )
      wire#w1
      Contact( "T-03_ChiliAwetan_2".Out_AV_CIP_Line )
      Coil( "IO_Valve_T03_Chili"."AV-03.01".AUT_OP )
   END_RUNG
   RUNG wire#w1
      Contact( "T-03_ChiliAwetan_2".Out_AV_CIP_Tank )
      Coil( "IO_Valve_T03_Chili"."AV-03.02".AUT_OP )
   END_RUNG
   RUNG wire#w1
      Contact( "T-03_ChiliAwetan_2".Out_AV_Outlet )
      wire#w2
      Coil( "IO_Valve_T03_Chili"."AV-03.03".AUT_OP )
   END_RUNG
   RUNG wire#w1
      Contact( "General Preparation"."Tipper 2"."CIP Request" )
      Contact( "General Preparation"."Tipper 2"."CIP Enable_T-03 Cmd" )
      Contact( "CIP_to_Mix".CIP_RequestOK.Osa_CIP_RequestOK )
   END_RUNG wire#w2
   RUNG wire#w1
      Contact( "T-03_ChiliAwetan_2".Out_AV_CIP_Tank )
      wire#w3
      Coil( "IO_Valve_T03_Chili"."AV-03.04".AUT_OP )
   END_RUNG
   RUNG wire#w1
      Contact( "General Preparation"."Tipper 2"."CIP Request" )
      Contact( "General Preparation"."Tipper 2"."CIP Enable_T-03 Cmd" )
      Contact( "CIP_to_Mix".CIP_RequestOK.Osa_CIP_RequestOK )
   END_RUNG wire#w3
   RUNG wire#w1
      Contact( "T-03_ChiliAwetan_2".Out_AV_CIP_Line )
      Coil( "IO_Valve_T03_Chili"."AV-03.05".AUT_OP )
   END_RUNG
   RUNG wire#w1
      Contact( "T-03_ChiliAwetan_2".Out_AV_Inload )
      wire#w4
      Coil( "IO_Valve_T03_Chili"."AV-03.06".AUT_OP )
   END_RUNG
   RUNG wire#w1
      Contact( "General Preparation"."Tipper 2"."CIP Request" )
      Contact( "General Preparation"."Tipper 2"."CIP Enable_T-03 Cmd" )
      Contact( "CIP_to_Mix".CIP_RequestOK.Osa_CIP_RequestOK )
   END_RUNG wire#w4
   RUNG wire#w1
      Contact( "T-03_ChiliAwetan_2".Out_AV_Transfer )
      Contact( "T-03_ChiliAwetan_2".IN_Dose_Header_2 )
      Coil( "IO_Valve_T03_Chili"."AV-03.11".AUT_OP )
   END_RUNG
   RUNG wire#w1
      Contact( "T-03_ChiliAwetan_2".Out_AV_Transfer )
      Contact( "T-03_ChiliAwetan_2".IN_Dose_Header_1 )
      Coil( "IO_Valve_T03_Chili"."AV-03.12".AUT_OP )
   END_RUNG
   RUNG wire#w1
      Contact( "T-03_ChiliAwetan_2".Out_AV_CIP_Line )
      Coil( "IO_Valve_T03_Chili"."AV-03.13".AUT_OP )
   END_RUNG
   // the same network as SCL:
   "IO_Valve_T03_Chili"."AV-03.01".AUT_OP := "AlwaysTRUE" AND "T-03_ChiliAwetan_2".Out_AV_CIP_Line;
   "IO_Valve_T03_Chili"."AV-03.02".AUT_OP := "AlwaysTRUE" AND "T-03_ChiliAwetan_2".Out_AV_CIP_Tank;
   "IO_Valve_T03_Chili"."AV-03.03".AUT_OP := "AlwaysTRUE" AND ("T-03_ChiliAwetan_2".Out_AV_Outlet OR ("General Preparation"."Tipper 2"."CIP Request" AND "General Preparation"."Tipper 2"."CIP Enable_T-03 Cmd" AND "CIP_to_Mix".CIP_RequestOK.Osa_CIP_RequestOK));
   "IO_Valve_T03_Chili"."AV-03.04".AUT_OP := "AlwaysTRUE" AND ("T-03_ChiliAwetan_2".Out_AV_CIP_Tank OR ("General Preparation"."Tipper 2"."CIP Request" AND "General Preparation"."Tipper 2"."CIP Enable_T-03 Cmd" AND "CIP_to_Mix".CIP_RequestOK.Osa_CIP_RequestOK));
   "IO_Valve_T03_Chili"."AV-03.05".AUT_OP := "AlwaysTRUE" AND "T-03_ChiliAwetan_2".Out_AV_CIP_Line;
   "IO_Valve_T03_Chili"."AV-03.06".AUT_OP := "AlwaysTRUE" AND ("T-03_ChiliAwetan_2".Out_AV_Inload OR ("General Preparation"."Tipper 2"."CIP Request" AND "General Preparation"."Tipper 2"."CIP Enable_T-03 Cmd" AND "CIP_to_Mix".CIP_RequestOK.Osa_CIP_RequestOK));
   "IO_Valve_T03_Chili"."AV-03.11".AUT_OP := "AlwaysTRUE" AND "T-03_ChiliAwetan_2".Out_AV_Transfer AND "T-03_ChiliAwetan_2".IN_Dose_Header_2;
   "IO_Valve_T03_Chili"."AV-03.12".AUT_OP := "AlwaysTRUE" AND "T-03_ChiliAwetan_2".Out_AV_Transfer AND "T-03_ChiliAwetan_2".IN_Dose_Header_1;
   "IO_Valve_T03_Chili"."AV-03.13".AUT_OP := "AlwaysTRUE" AND "T-03_ChiliAwetan_2".Out_AV_CIP_Line;
END_REGION

